	MW(WORD_WEAK := MesBlock_Temp[2][1], 	WORD_STRONG:= MesBlock_Temp[2][2], VAR_OUT:= MesDataExd.MesData.MesU12);		
	MW(WORD_WEAK := MesBlock_Temp[2][3], 	WORD_STRONG:= MesBlock_Temp[2][4], VAR_OUT:= MesDataExd.MesData.MesU23);
	MW(WORD_WEAK := MesBlock_Temp[2][5], 	WORD_STRONG:= MesBlock_Temp[2][6], VAR_OUT:= MesDataExd.MesData.MesU31);
	MW(WORD_WEAK := MesBlock_Temp[2][7], 	WORD_STRONG:= MesBlock_Temp[2][8], VAR_OUT:= MesDataExd.MesData.MesU);		// Seule donnée valide en monophasée. Il faut d'ailleur inverser les words strongs et word weak quand on passe le settings de triphasé à monophasé . 
	MW(WORD_WEAK := MesBlock_Temp[2][9], 	WORD_STRONG:= MesBlock_Temp[2][10], VAR_OUT:= MesDataExd.MesData.MesV1);
	MW(WORD_WEAK := MesBlock_Temp[2][11], WORD_STRONG := MesBlock_Temp[2][12], VAR_OUT:= MesDataExd.MesData.MesV2);
	MW(WORD_WEAK := MesBlock_Temp[2][13], WORD_STRONG := MesBlock_Temp[2][14], VAR_OUT:= MesDataExd.MesData.MesV3);
	MW(WORD_WEAK := MesBlock_Temp[2][17], WORD_STRONG := MesBlock_Temp[2][18], VAR_OUT:= MesDataExd.MesData.MesV);
	
	MW( WORD_STRONG:= MesBlock_Temp[3][1], 	WORD_WEAK := MesBlock_Temp[3][2], VAR_OUT:= MesDataExd.MesData.MesP1);
	MW( WORD_STRONG:= MesBlock_Temp[3][3], 	WORD_WEAK := MesBlock_Temp[3][4], VAR_OUT:= MesDataExd.MesData.MesP2);
	MW( WORD_STRONG:= MesBlock_Temp[3][5], 	WORD_WEAK := MesBlock_Temp[3][6], VAR_OUT:= MesDataExd.MesData.MesP3);
	MW( WORD_STRONG:= MesBlock_Temp[3][7], 	WORD_WEAK := MesBlock_Temp[3][8], VAR_OUT:= MesDataExd.MesData.MesP);
	
	MW( WORD_STRONG:= MesBlock_Temp[3][9], 	WORD_WEAK := MesBlock_Temp[3][10], VAR_OUT:= MesDataExd.MesData.MesQ1);
	MW( WORD_STRONG:= MesBlock_Temp[3][11], 	WORD_WEAK := MesBlock_Temp[3][12], VAR_OUT:= MesDataExd.MesData.MesQ2);
	MW( WORD_STRONG:= MesBlock_Temp[3][13], 	WORD_WEAK := MesBlock_Temp[3][14], VAR_OUT:= MesDataExd.MesData.MesQ3);
	MW( WORD_STRONG:= MesBlock_Temp[3][15], 	WORD_WEAK := MesBlock_Temp[3][16], VAR_OUT:= MesDataExd.MesData.MesQ);
	MW( WORD_STRONG:= MesBlock_Temp[3][23], 	WORD_WEAK := MesBlock_Temp[3][24], VAR_OUT:= MesDataExd.MesData.MesS);
	
	MW( WORD_STRONG:= MesBlock_Temp[4][1], 	WORD_WEAK := MesBlock_Temp[4][2], VAR_OUT:= MesDataExd.MesData.MesTanPhi);
	MW( WORD_STRONG:= MesBlock_Temp[4][3], 	WORD_WEAK := MesBlock_Temp[4][4], VAR_OUT:= MesDataExd.MesData.MesFreq);
	
	MW2( WORD_STRONG:= MesBlock_Temp[5][3], 	WORD_WEAK := MesBlock_Temp[5][4], VAR_OUT := MesDataExd.MesData.MesEActCons,SIZE:=2,FIX:=3);
	MW2( WORD_STRONG:= MesBlock_Temp[5][7], 	WORD_WEAK := MesBlock_Temp[5][8], VAR_OUT := MesDataExd.MesData.MesEActProd,SIZE:=2,FIX:=3);
	MW2( WORD_STRONG:= MesBlock_Temp[5][19], 	WORD_WEAK := MesBlock_Temp[5][20], VAR_OUT := MesDataExd.MesData.MesEReactProd,SIZE:=2,FIX:=3);
	MW2( WORD_STRONG:= MesBlock_Temp[5][23], 	WORD_WEAK := MesBlock_Temp[5][24], VAR_OUT := MesDataExd.MesData.MesEReactCons,SIZE:=2,FIX:=3);
	
	
	//MW( WORD_STRONG:= MesBlock_Temp[4][3], 	WORD_WEAK := MesBlock_Temp[4][4],	SIGNED:=TRUE, FIX:=0 , SIZE:=2, VAR_OUT := MesDataExd.MesData.MesFreq);
	//MW( WORD_STRONG:= MesBlock_Temp[5][1], 	WORD_WEAK := MesBlock_Temp[5][2],	SIGNED:=TRUE, FIX:=0 , SIZE:=2, VAR_OUT := MesDataExd.MesData.MesEActProd);
	//MW( WORD_STRONG:= MesBlock_Temp[5][3], 	WORD_WEAK := MesBlock_Temp[5][4],	SIGNED:=TRUE, FIX:=0 , SIZE:=2, VAR_OUT := MesDataExd.MesData.MesEActCons);
	//MW( WORD_STRONG:= MesBlock_Temp[5][5], 	WORD_WEAK := MesBlock_Temp[5][6],	SIGNED:=TRUE, FIX:=0 , SIZE:=2, VAR_OUT := MesDataExd.MesData.MesEReactProd);
	//MW( WORD_STRONG:= MesBlock_Temp[5][7], 	WORD_WEAK := MesBlock_Temp[5][8],	SIGNED:=TRUE, FIX:=0 , SIZE:=2, VAR_OUT := MesDataExd.MesData.MesEReactCons);
END_IF
END_METHOD

END_FUNCTION_BLOCK

// ---- 01_Equipement_Library/Datalogger/FB_Datalogger_PPCVerrerie.TcPOU
FUNCTION_BLOCK FB_Datalogger_PPCVerrerie	EXTENDS FB_Datalogger_Base	// Data from PPC ( MV + HV )
VAR_INPUT PERSISTENT
	// Parameters of the Object (instance specific) 
	ParamTempoComAlarm			: TIME 			:= T#10S ; 						// (s) Config : Tempo to detect LOC Alarm
	{attribute 'OPC.UA.DA' := '1'} 
	ParamClockReadTime 			: TIME 			:= TIME#200MS;	  				// (Time) Read Modbus Frequency.  
	ParamTimeout				: TIME  		:= T#2S ;			  			// (Time) Timeout for modbus reading
	ParamIPAdr : STRING := '192.168.1.2'; // IP Address for Modbus Requests 
END_VAR
VAR_INPUT
	IN_CmdToggleRead			: BOOL ;
	IN_CmdReset_L				: BOOL  ; // Reset Order .
	
	MesDataExd	AT %Q*				: Datalogger_PPCVerrerie;
	
END_VAR
VAR

	
	//M_ALARMMANAGEMENT VARIABLES//
	TON_ComAlarm				: TON ; 												// Tempo before detecting loss of communication. 
	TON_ComWarning				: TON ; 												// Tempo before detecting loss of one frame.   
	
	MesComWarning				: BOOL ; 												// True if bad communication .
	
	// M_EXECUTE VARIABLES //
	
	TP1							: TP ; 												// (NA) Tempo to define Modbus Reading Frequency  
	
    Trig_Cmd_Read				: R_TRIG;                       

	// Modbus Read Variables
	
	FB_ModbusReadAI : ARRAY[1..2] OF FB_ModbusRead;
	FB_ModbusReadDI : ARRAY[1..2] OF FB_ModbusReadCoils;
	
	ClockRead					AT %Q*		: BOOL ;
	
	// Temp Blocks Filled by Requests
	
	AI_List_1 				: ARRAY[1..128] OF WORD;
	AI_List_2 				: ARRAY[1..128] OF WORD;
	DI_List_1 				: ARRAY[1..2048] OF BOOL;
	DI_List_2 				: ARRAY[1..2048] OF BOOL;
	
	
	
END_VAR

METHOD M_AlarmManagement : BOOL
VAR_INPUT
END_VAR
//////////////////
// Digiware measurement tool alarm and warning management
/////////////////

VAR 
	// Method local variables (reinitialized at each cycle) 
	FB_AlarmCodeManager			: FB_AlarmCodeManager ; 
	
	ComWarning					: BOOL;			// Error in one of the Modbus Requests
	ComAlarm					: BOOL;			// Error in all Modbus Requests
	
END_VAR
ComWarning 	:= FB_ModbusReadAI[1].ModbusReadAlarm OR FB_ModbusReadAI[2].ModbusReadAlarm OR FB_ModbusReadDI[1].ModbusReadAlarm OR FB_ModbusReadDI[2].ModbusReadAlarm;
ComAlarm 	:= FB_ModbusReadAI[1].ModbusReadAlarm AND FB_ModbusReadAI[2].ModbusReadAlarm AND FB_ModbusReadDI[1].ModbusReadAlarm AND FB_ModbusReadDI[2].ModbusReadAlarm;
	
TON_ComAlarm(IN:= ComAlarm , PT:= ParamTempoComAlarm, Q= MesDataExd.MesData.MesAlarmCom) ;	
TON_ComWarning(IN:= ComWarning  , PT:= ParamTempoComAlarm, Q=>MesComWarning) ;

//	General com alarm : All the read FB fucked up


// ALARM CODES //
	FB_AlarmCodeManager(
		bAlarm1			:= MesDataExd.MesData.MesAlarmCom , 						// Communication Alarm #COM
		bAlarm2			:= MesDataExd.MesData.Transfo_225kV.MesWarning_TempLevel1,	// Transfo_225kV : Img Therm 1
		bAlarm3			:= MesDataExd.MesData.Transfo_225kV.MesWarning_TempLevel2,	// Transfo_225kV : Img Therm 2
		bAlarm4			:= MesDataExd.MesData.Transfo_225kV.MesDataExd.MesData.MesAlarmTemp,	// Transfo_225kV : Trigger Temp Oil
		bAlarm5			:= MesDataExd.MesData.Transfo_225kV.MesAlarm_TapChanger ,	// Transfo 225kV : Defaillance Regleur
		bAlarm6			:= MesDataExd.MesData.Mes20kVCourNeutCuveTempTrigger,		// 20 kV Courant Neutre Cuve : Temp Trigger
		bAlarm7			:= MesDataExd.MesData.Mes20kVCourNeutCuveGazDischarge,		// 20 kV Courant Neutre Cuve : Gaz Discharge
		bAlarm8			:= MesDataExd.MesData.Mes20kVCourNeutCuvePressure,			// 20 kV Courant Neutre Cuve : Pressure
		bAlarm9			:= MesDataExd.MesData.Transfo_225kV.MesDataExd.MesData.MesAlarmGas,	// Transfo 225kV : Trigger BuchHolz
		bAlarm10		:= MesDataExd.MesData.Transfo_225kV.MesTrigger_Deletion,	// Transfo_225kV : Trigger Deletion
		bAlarm11		:= MesDataExd.MesData.Transfo_225kV.MesAlarm_OilLevel,      // Transfo_225kV : Alarm Oil level
		bAlarm12		:= MesDataExd.MesData.DS.MesAlarmState,          		// DS : Doors Open          
		bAlarm13		:= MesDataExd.MesData.FSS.MesAlarmFire,			        // FSS : Fire Alarm
		bAlarm14		:= MesDataExd.MesData.MesLocalRemoteOperation, 			// Local/Remote Operation
		bAlarm15		:= MesDataExd.MesData.ES.MesAlarmState,         	 	// ES : Emergency Stop			 
		wAlarmCode		=>MesDataExd.MesData.MesAlarmCode1);

	FB_AlarmCodeManager(	
		bAlarm1			:= MesDataExd.MesData.ProtectRelay_Transfo225kV.MesAlarm_DiscordSectLigneHTB,	//	ProtectRelay_Transfo_225kV :	Alarm Discord Sect Ligne HTB
		bAlarm2			:= MesDataExd.MesData.ProtectRelay_Transfo225kV.MesAlarm_DiscordSectMaltHTB ,   //  ProtectRelay_Transfo_225kV : Alarm Discord Sect Malt HTB 
		bAlarm3			:= MesDataExd.MesData.ProtectRelay_Transfo225kV.MesAlarm_DiscordSectDisjHTB ,   //  ProtectRelay_Transfo_225kV : Alarm Discord Sect Disj HTB 
		bAlarm4			:= MesDataExd.MesData.ProtectRelay_Transfo225kV.MesAlarm_TeleCondamne       ,   //  ProtectRelay_Transfo_225kV : Alarm Tele Condamne       
		bAlarm5			:= MesDataExd.MesData.ProtectRelay_Transfo225kV.MesAlarm_DeTeleCondamne     ,   //  ProtectRelay_Transfo_225kV : Alarm DeTele Condamne     
		bAlarm6			:= MesDataExd.MesData.ProtectRelay_Transfo225kV.MesAlarm_DiscordTeleCondamne,   //  ProtectRelay_Transfo_225kV : Alarm Discord Tele Condamne
		bAlarm7			:= MesDataExd.MesData.ProtectRelay_Transfo225kV.MesDataExd.MesData.MesAlarmImax        ,   //  ProtectRelay_Transfo_225kV : Alarm Imax
		bAlarm8			:= MesDataExd.MesData.ProtectRelay_Transfo225kV.MesAlarm_IoMaxCoteProd      ,   //  ProtectRelay_Transfo_225kV : Alarm Io Max Cote Prod
		bAlarm9			:= MesDataExd.MesData.ProtectRelay_Transfo225kV.MesDataExd.MesData.MesAlarmUmin        ,   //  ProtectRelay_Transfo_225kV : Alarm U min
		bAlarm10		:= MesDataExd.MesData.ProtectRelay_Transfo225kV.MesDataExd.MesData.MesAlarmUmin_Long   ,   //  ProtectRelay_Transfo_225kV : Alarm U min Long
		bAlarm11		:= MesDataExd.MesData.ProtectRelay_Transfo225kV.MesAlarmUMax                ,   //  ProtectRelay_Transfo_225kV : Alarm U max
		bAlarm12		:= MesDataExd.MesData.ProtectRelay_Transfo225kV.MesAlarmUMax_Long           ,   //  ProtectRelay_Transfo_225kV : Alarm U max Long
		bAlarm13		:= MesDataExd.MesData.ProtectRelay_Transfo225kV.MesAlarm_PhaseRpt           ,   //  ProtectRelay_Transfo_225kV : Alarm Phase Rpt
		bAlarm14		:= MesDataExd.MesData.ProtectRelay_Transfo225kV.MesAlarm_ImgTherm     		,	//	ProtectRelay_Transfo_225kV : Alarm Img Therm
		bAlarm15		:= MesDataExd.MesData.ProtectRelay_Transfo225kV.MesAlarm_DifferTransfo		,	//  ProtectRelay_Transfo_225kV : Alarm Differ Transfo
		wAlarmCode		=>MesDataExd.MesData.MesAlarmCode2);	


	FB_AlarmCodeManager(	
		bAlarm1			:= MesDataExd.MesData.ProtectRelay_Transfo225kV.MesAlarm_FreqMax ,	// ProtectRelay_Transfo_225kV : Alarm Freq Max
		bAlarm2			:= MesDataExd.MesData.ProtectRelay_Transfo225kV.MesAlarm_FreqMin ,  // ProtectRelay_Transfo_225kV : Alarm Freq Min
		bAlarm3			:= MesDataExd.MesData.MainHVCB.MesDataExd.MesData.MesClosed ,					// MainHVCB : Closed 
		bAlarm4			:= MesDataExd.MesData.MainHVCB.MesAlarm_SF6      ,					// MainHVCB : Alarm SF6
		bAlarm5			:= MesDataExd.MesData.MainHVCB.MesAlarm_Disarmed ,					// MainHVCB : Alarm Disarmed
		bAlarm6			:= MesDataExd.MesData.MainHVCB.MesComutLocal     ,					// MainHVCB : Comut Local
		bAlarm7			:= MesDataExd.MesData.Transfo_225kV.MesTransfoRefrigLocal,    		// Transfo_225kV : Transfo Refrig Local
		bAlarm8			:= MesDataExd.MesData.Transfo_225kV.MesTrigger_NonReturnValve,      // Transfo_225kV : Trigger Non Return Valve
		bAlarm9			:= MesDataExd.MesData.Transfo_225kV.MesTrigger_ProtectRelay,        // Transfo_225kV : Trigger Protect Relay
		bAlarm10		:= MesDataExd.MesData.Transfo_Aux.MesDataExd.MesData.MesAlarmTemp,				// Transfo_Aux : Alarm Temp
		bAlarm11		:= MesDataExd.MesData.Transfo_Aux.MesDataExd.MesData.MesAlarmGas,              // Transfo_Aux : Alarm Gas
		bAlarm12		:= MesDataExd.MesData.Transfo_Aux.MesDataExd.MesData.MesAlarmOilLevel,         // Transfo_Aux : Alarm Pressure
		bAlarm13		:= MesDataExd.MesData.MesAuxTransfoMeltingFusesContact,			// Transfo_Aux : Melting Fuses Contact     
		bAlarm14		:= MesDataExd.MesData.MesAuxTransfoSwitchGear,                     // Transfo_Aux : Transfo Switch Gear
		bAlarm15		:=FALSE,
		wAlarmCode		=>MesDataExd.MesData.MesAlarmCode3);			
		
		
// WARNING CODES //
	FB_AlarmCodeManager(		
		bAlarm1			:=MesComWarning	,				 							// Communication Warning
		bAlarm2			:= MesDataExd.MesData.ProtectRelay_MainHVCB.MesAlarm_Phase1 , 			// ProtectRelay_MainHVCB : Default Phase 1       
		bAlarm3			:= MesDataExd.MesData.ProtectRelay_MainHVCB.MesAlarm_Phase2 , 			// ProtectRelay_MainHVCB : Default Phase 2       
		bAlarm4			:= MesDataExd.MesData.ProtectRelay_MainHVCB.MesAlarm_Phase3 , 			// ProtectRelay_MainHVCB : Default Phase 3       
		bAlarm5			:= MesDataExd.MesData.ProtectRelay_MainHVCB.MesAlarm_PhaseRpt , 		// ProtectRelay_MainHVCB : Default Phase Rpt      
		bAlarm6			:= MesDataExd.MesData.ProtectRelay_MainHVCB.MesAlarm_Ground , 			// ProtectRelay_MainHVCB : Default Phase Ground        
		bAlarm7			:= MesDataExd.MesData.ProtectRelay_MainHVCB.MesAlarm_GroundRpt , 		// ProtectRelay_MainHVCB : Default Phase Ground Rpt     
		bAlarm8			:= MesDataExd.MesData.ProtectRelay_MainHVCB.MesAlarm_MaxUInverse , 		// ProtectRelay_MainHVCB : Default Max U Inverse   
		bAlarm9			:= MesDataExd.MesData.ProtectRelay_MainHVCB.MesAlarm_MaxP , 			// ProtectRelay_MainHVCB : Default Max P
		bAlarm10		:= MesDataExd.MesData.ProtectRelay_MainHVCB.MesAlarm_CB , 				// ProtectRelay_MainHVCB : Default Circuit Breaker
		bAlarm11		:= MesDataExd.MesData.ProtectRelay_MainHVCB.MesAlarm_Watchdog , 		// ProtectRelay_MainHVCB : Default Watchdog     
		bAlarm12		:= MesDataExd.MesData.ProtectRelay_MainHVCB.MesDataExd.MesData.MesAlarmTCS  , 		// ProtectRelay_MainHVCB : Default Major        
		bAlarm13		:= MesDataExd.MesData.ProtectRelay_Transfo225kV.MesAlarm_PhaseRpt ,		// ProtectRelay_Transfo225kV : Default Phase Rpt
		bAlarm14		:= MesDataExd.MesData.ProtectRelay_Transfo225kV.MesAlarm_ImgTherm , 	// ProtectRelay_Transfo225kV : Default img Therm
		bAlarm15		:= MesDataExd.MesData.MainHVCB.MesAlarm_ArmingMotor , 					// MainHVCB : Default Arming Motor
		wAlarmCode		=>MesDataExd.MesData.MesWarningCode1);

	FB_AlarmCodeManager(		
		bAlarm1			:= MesDataExd.MesData.MainHVCB.MesAlarm_230V, 							// MainHVCB : Default Aux 230 Vac				 
		bAlarm2			:= MesDataExd.MesData.MainHVCB.MesAlarmPwr, 							// MainHVCB : Default Alim Bobine
		bAlarm3			:= MesDataExd.MesData.Transfo_225kV.MesWarningGas, 						// Transfo_225kV : Buchholz Gas Warning
		bAlarm4			:= MesDataExd.MesData.Transfo_225kV.MesDataExd.MesData.MesWarningTemp, 			// Transfo_225kV : Temperature Warning
		bAlarm5			:= MesDataExd.MesData.ProtectRelay_Transfo225kV.MesDataExd.MesData.MesAlarmTCS , 	// ProtectRelay_Transfo225kV : Major Default
		bAlarm6			:= MesDataExd.MesData.ProtectRelay_Transfo225kV.MesWarning_ImgTherm , 	// ProtectRelay_Transfo225kV : Warning Img Therm
		bAlarm7			:= MesDataExd.MesData.TapChanger.MesAlarm,								// 225 kV Regleur : Default
		bAlarm8			:= MesDataExd.MesData.TapChanger.MesAlarm_Discordance, 					// 225 kV Regleur : Default Discordance
		bAlarm9			:= MesDataExd.MesData.ProtectRelay_MainMVCB.MesAlarm_Phase1, 			// Protection Relay Main MVCB : Default Phase 1
		bAlarm10		:= MesDataExd.MesData.ProtectRelay_MainMVCB.MesAlarm_Phase2, 			// Protection Relay Main MVCB : Default Phase 2
		bAlarm11		:= MesDataExd.MesData.ProtectRelay_MainMVCB.MesAlarm_CB, 				// Protection Relay Main MVCB : Default Circuit Breaker
		bAlarm12		:=FALSE , 													//
		bAlarm13		:= MesDataExd.MesData.MainMVCB.MesTripped 	, 							// Main MVCB : Tripped
		bAlarm14		:= MesDataExd.MesData.ProtectRelay_MainMVCB.MesDataExd.MesData.MesAlarmTCS , 		// Protection Relay Main MVCB : Alarm TCS
		bAlarm15		:= MesDataExd.MesData.ProtectRelay_MainMVCB.MesDataExd.MesData.MesWatchdog,		// Protection Relay Main MVCB : Watchdog
		wAlarmCode		=>MesDataExd.MesData.MesWarningCode2);		

	FB_AlarmCodeManager(		
		bAlarm1			:= MesDataExd.MesData.ProtectRelay_FeederMVCB[1].MesDataExd.MesData.MesAlarmImax, 							//  ProtectRelay_FeederMVCB Midi Max I Alarm
		bAlarm2			:= MesDataExd.MesData.ProtectRelay_FeederMVCB[1].MesAlarm_MaxP ,								//  ProtectRelay_FeederMVCB Midi Max P Alarm 
		bAlarm3			:= MesDataExd.MesData.ProtectRelay_FeederMVCB[1].MesAlarm_Ground , 								//  ProtectRelay_FeederMVCB Midi Ground Alarm
		bAlarm4			:= MesDataExd.MesData.ProtectRelay_FeederMVCB[1].MesAlarm_CablesOvercharge, 					//	ProtectRelay_FeederMVCB Midi Cables Overcharge
		bAlarm5			:= MesDataExd.MesData.ProtectRelay_FeederMVCB[1].MesAlarm_FaultFrom225kV, 						//  ProtectRelay_FeederMVCB Midi Fault From 225 kV   
		bAlarm6			:= MesDataExd.MesData.ProtectRelay_FeederMVCB[1].MesDataExd.MesData.MesAlarmTCS , 							//  ProtectRelay_FeederMVCB Midi Default Major       
		bAlarm7			:= MesDataExd.MesData.ProtectRelay_FeederMVCB[2].MesDataExd.MesData.MesAlarmImax, 	 						//  ProtectRelay_FeederMVCB Plat Max I Alarm      
		bAlarm8			:= MesDataExd.MesData.ProtectRelay_FeederMVCB[2].MesAlarm_MaxP ,			     				//  ProtectRelay_FeederMVCB Plat Max P Alarm        
		bAlarm9			:= MesDataExd.MesData.ProtectRelay_FeederMVCB[2].MesAlarm_Ground , 		   						//  ProtectRelay_FeederMVCB Plat Ground Alarm          
		bAlarm10		:= MesDataExd.MesData.ProtectRelay_FeederMVCB[2].MesAlarm_CablesOvercharge, 					//  ProtectRelay_FeederMVCB Plat Cables Overcharge 
		bAlarm11		:= MesDataExd.MesData.ProtectRelay_FeederMVCB[2].MesAlarm_FaultFrom225kV, 	 					//  ProtectRelay_FeederMVCB Plat Fault From 225 kV    
		bAlarm12		:= MesDataExd.MesData.ProtectRelay_FeederMVCB[2].MesDataExd.MesData.MesAlarmTCS,				 			//  ProtectRelay_FeederMVCB Plat Default Major                  
		bAlarm13		:=FALSE,   //
		bAlarm14		:=FALSE,   //
		bAlarm15		:=FALSE,   //
		wAlarmCode		=>MesDataExd.MesData.MesWarningCode3);

	FB_AlarmCodeManager(		
		bAlarm1			:= MesDataExd.MesData.Mes20kVCourNeutCuveDefaultMasseCuve1,			//	 20 kV Courant Neutre Cuve Default Masse 1
		bAlarm2			:= MesDataExd.MesData.Mes20kVCourNeutCuveDefaultMasseCuve2,			//	 20 kV Courant Neutre Cuve Default Masse 2
		bAlarm3			:= MesDataExd.MesData.Mes20kVCourNeutCuveDefaultGround,				//	 20 kV Courant Neutre Cuve Default Ground 
		bAlarm4			:= MesDataExd.MesData.Mes20kVCourNeutCuveTempAlarm,					//	 20 kV Courant Neutre Cuve Temp  
		bAlarm5			:= MesDataExd.MesData.MesAuxBt400VDefaultPermut, 					//	 Aux Bt 400 V  : Default Permut 
		bAlarm6			:= MesDataExd.MesData.UPS_CE.MesAlarm_Batt, 			      		//	 UPC CE : Default Batt
		bAlarm7			:= MesDataExd.MesData.UPS_CE.MesDataExd.MesData.MesAlarmState, 				//	 UPC CE : Default Redress
		bAlarm8			:= MesDataExd.MesData.UPS_CE.MesAlarm_IsolBatt,		    			//   UPC CE : Default Isol Batt
		bAlarm9			:= MesDataExd.MesData.UPS_TCM.MesAlarm_Batt,			      		//   UPC TCM : Default Batt
		bAlarm10		:= MesDataExd.MesData.UPS_TCM.MesDataExd.MesData.MesAlarmState,	 			//	 UPC TCM : Default Redress
		bAlarm11		:= MesDataExd.MesData.MesAuxBtDefaultInverter, 						//	 Aux Bt : Default Inverter
		bAlarm12		:= MesDataExd.MesData.MesAuxBtSyntDefaultDistrib48VccJdb, 			//	 Aux Bt Synt : Default Distrib 48 Vcc Jdb
		bAlarm13		:= MesDataExd.MesData.MesAuxBtSyntDefaultDistrib48VccLocker, 		//	 Aux Bt Synt : Default Distrib 48 Vcc Locker
		bAlarm14		:=FALSE, //
		bAlarm15		:=FALSE, //
		wAlarmCode		=>MesDataExd.MesData.MesWarningCode4);		
		
	FB_AlarmCodeManager(		
		bAlarm1			:= MesDataExd.MesData.Mes20kVCourNeutCuveMaxIexp2,	//	 20 kV Courant Neutre Cuve Default Max I Exp 2
		bAlarm2			:= MesDataExd.MesData.Mes20kVCourNeutCuveMaxIexp4,  //	 20 kV Courant Neutre Cuve Default Max I Exp 4
		bAlarm3			:= MesDataExd.MesData.Mes20kVCourNeutCuveMaxI0exp4, //	 20 kV Courant Neutre Cuve Default Max I0 Exp 4
		bAlarm4			:= MesDataExd.MesData.ProtectRelay_FeederMVCB[1].MesDataExd.MesData.MesTripped, // ProtectRelay_FeederMVCB Midi Tripped
		bAlarm5			:= MesDataExd.MesData.ProtectRelay_FeederMVCB[2].MesDataExd.MesData.MesTripped, // ProtectRelay_FeederMVCB Plat Tripped
		bAlarm6			:= MesDataExd.MesData.MesAuxHTSect225kV		,					//	Aux HT : Sect 225 kV
		bAlarm7			:= MesDataExd.MesData.MesAuxHtSmaltHTBOpen	,                   //	Aux HT : Malt HTB Open
		bAlarm8			:= MesDataExd.MesData.MesAuxHtFusionFuseMeasures225kV	,       //	Aux HT : Fusion Fuse Measures 225 kV
		bAlarm9			:= MesDataExd.MesData.MesAuxHtFusionFuseProtect225kV	,       //  Aux HT : Fusion Fuse Protect 225 kV
		bAlarm10		:= MesDataExd.MesData.MesAuxHtFusionFuseCountRte225kV	,       //	Aux HT : Fusion Fuse Count Rte 225 kV
		bAlarm11		:= MesDataExd.MesData.MesAuxHtShortCircuitCurrentProtectCcp2,   //  Aux HT : Short Circuit Current Protect Ccp2
		bAlarm12		:= MesDataExd.MesData.MesAuxHtDisjCount20kVOpen		,           //	Aux HT : Disj Count 20kV Open
		bAlarm13		:= MesDataExd.MesData.MesAuxHtDisjRefVoltage20kVOpen,			//  Aux HT : Disj Ref Voltage 20kV Open
		bAlarm14		:= MesDataExd.MesData.MesAuxHtShortCircuitCurrentProtectCcp3, 	//	Aux HT : Short Circuit Current Protect Ccp3
		bAlarm15		:= MesDataExd.MesData.MesAuxBtTriggerGeneralDisj, 				//  Aux BT : Trigger General Disj
		wAlarmCode		=>MesDataExd.MesData.MesWarningCode5);
		
	FB_AlarmCodeManager(		
		bAlarm1			:= MesDataExd.MesData.Mes20kVCourNeutCuveMaxIexp2,	//	 20 kV Courant Neutre Cuve Default Max I Exp 2
		bAlarm2			:= MesDataExd.MesData.Mes20kVCourNeutCuveMaxIexp4,  //	 20 kV Courant Neutre Cuve Default Max I Exp 4
		bAlarm3			:= MesDataExd.MesData.Mes20kVCourNeutCuveMaxI0exp4, //	 20 kV Courant Neutre Cuve Default Max I0 Exp 4
		bAlarm4			:= MesDataExd.MesData.ProtectRelay_FeederMVCB[1].MesDataExd.MesData.MesTripped, // ProtectRelay_FeederMVCB Midi Tripped
		bAlarm5			:= MesDataExd.MesData.ProtectRelay_FeederMVCB[2].MesDataExd.MesData.MesTripped, // ProtectRelay_FeederMVCB Plat Tripped
		bAlarm6			:= MesDataExd.MesData.MesAuxHTSect225kV		,					//	Aux HT : Sect 225 kV
		bAlarm7			:= MesDataExd.MesData.MesAuxHtSmaltHTBOpen	,                   //	Aux HT : Malt HTB Open
		bAlarm8			:= MesDataExd.MesData.MesAuxHtFusionFuseMeasures225kV	,       //	Aux HT : Fusion Fuse Measures 225 kV
		bAlarm9			:= MesDataExd.MesData.MesAuxHtFusionFuseProtect225kV	,       //  Aux HT : Fusion Fuse Protect 225 kV
		bAlarm10		:= MesDataExd.MesData.MesAuxHtFusionFuseCountRte225kV	,       //	Aux HT : Fusion Fuse Count Rte 225 kV
		bAlarm11		:= MesDataExd.MesData.MesAuxHtShortCircuitCurrentProtectCcp2,   //  Aux HT : Short Circuit Current Protect Ccp2
		bAlarm12		:= MesDataExd.MesData.MesAuxHtDisjCount20kVOpen		,           //	Aux HT : Disj Count 20kV Open
		bAlarm13		:= MesDataExd.MesData.MesAuxHtDisjRefVoltage20kVOpen,			//  Aux HT : Disj Ref Voltage 20kV Open
		bAlarm14		:= MesDataExd.MesData.MesAuxHtShortCircuitCurrentProtectCcp3, 	//	Aux HT : Short Circuit Current Protect Ccp3
		bAlarm15		:= MesDataExd.MesData.MesAuxBtTriggerGeneralDisj, 				//  Aux BT : Trigger General Disj
		wAlarmCode		=>MesDataExd.MesData.MesWarningCode6);
		
		
// EVENT CODE //
	FB_AlarmCodeManager(
		bAlarm1			:= MesDataExd.MesData.MesAuxBt400VManqueAC			 ,  		// Aux BT 400 V : Manque AC     
		bAlarm2			:= MesDataExd.MesData.MesAuxBt400VDecltAntenneScada	 ,  		// Aux BT 400 V : Declt Antenne Scada
		bAlarm3			:= MesDataExd.MesData.MesAuxBt400VDecltAntennePrio	 ,  		// Aux BT 400 V : Declt Antenne Prio
		bAlarm4			:= MesDataExd.MesData.MesAuxBt400VVoltageLossNormalAlim	, 		// Aux BT 400 V : Voltage Loss Normal Alim
		bAlarm5			:= MesDataExd.MesData.MesAuxBt400VVoltageLossSecoursAlim,   	// Aux BT 400 V : Voltage Loss Secours Alim
		bAlarm6			:= MesDataExd.MesData.MesAuxBt400VDefaultPermut	,           	// Aux BT 400 V : Default Permut 
		bAlarm7			:= MesDataExd.MesData.TapChanger.MesModeAuto, 					// 225 kV Regleur :	Mode Auto
		bAlarm8			:= MesDataExd.MesData.TapChanger.MesModeManual,                 // 225 kV Regleur :	Mode Manual                                                                                                                                                                                              
		bAlarm9			:= MesDataExd.MesData.TapChanger.MesState_ManoeuverAuthorized, 	// 225 kV Regleur :	State Manoeuver Authorized
		bAlarm10		:= MesDataExd.MesData.TapChanger.MesAlarm_NoOutletDetected, 	// 225 kV Regleur :	No Outlet Detected	
		bAlarm11		:= MesDataExd.MesData.ProtectRelay_MainHVCB.OUT_CmdOpen , 		// ProtectRelay_MainHVCB : Cmd Open
		bAlarm12		:= MesDataExd.MesData.ProtectRelay_MainHVCB.OUT_CmdClose,       // ProtectRelay_MainHVCB : Cmd Close
		bAlarm13		:= MesDataExd.MesData.ProtectRelay_MainMVCB.OUT_CmdOpen ,       // ProtectRelay_MainMVCB : Cmd Open
		bAlarm14		:= MesDataExd.MesData.ProtectRelay_MainMVCB.OUT_CmdClose,       // ProtectRelay_MainMVCB : Cmd Close
		bAlarm15		:=FALSE, 
		wAlarmCode		=>MesDataExd.MesData.MesEventCode1);
	
	FB_AlarmCodeManager(	
		bAlarm1			:= MesDataExd.MesData.ProtectRelay_FeederMVCB[1].OUT_CmdOpen , 	// ProtectRelay_FeederMVCB Midi : Cmd Open
		bAlarm2			:= MesDataExd.MesData.ProtectRelay_FeederMVCB[1].OUT_CmdClose,     // ProtectRelay_FeederMVCB Midi  : Cmd Close
		bAlarm3			:= MesDataExd.MesData.ProtectRelay_FeederMVCB[2].OUT_CmdOpen  ,    // ProtectRelay_FeederMVCB Plat  : Cmd Open
		bAlarm4			:= MesDataExd.MesData.ProtectRelay_FeederMVCB[2].OUT_CmdClose ,	// ProtectRelay_FeederMVCB Plat  : Cmd Close
		bAlarm5			:= MesDataExd.MesData.TapChanger.OUT_CmdRampUp,					// 225 kV Regleur : Cmd Ramp Up
		bAlarm6			:= MesDataExd.MesData.TapChanger.OUT_CmdRampDown ,                 // 225 kV Regleur :	Cmd Ramp Down
		bAlarm7			:= MesDataExd.MesData.MesAuxHtOpenSectLine225kV	 ,				// Aux Ht : Sect Line 225 kV Open
		bAlarm8			:= MesDataExd.MesData.MesAuxHtCloseSectLine225kV	,               // Aux Ht : Sect Line 225 kV Close
		bAlarm9			:= MesDataExd.MesData.MesAuxHtTeleCondamnSl225kV	 ,				// Aux Ht : Tele Condamn Sl 225 kV 
		bAlarm10		:= MesDataExd.MesData.MesAuxHtDeTeleCondamnSl225kV,       		// Aux Ht : DeTele Condamn Sl 225 kV
		bAlarm11		:= MesDataExd.MesData.MesAuxHtTelecommandeRelestActif ,			// Aux Ht : Telecommande Relest Actif
		bAlarm12		:= MesDataExd.MesData.MesAuxHtTelecommandeRelestPassif,           // Aux Ht : Telecommande Relest Passif
		bAlarm13		:= FALSE,
		bAlarm14		:= FALSE,
		bAlarm15		:= FALSE,
		wAlarmCode		=>MesDataExd.MesData.MesEventCode2);	
		
		
	FB_AlarmCodeManager(
		bAlarm1			:= MesDataExd.MesData.MesAuxHtOpenSectMalt,				// Aux Ht Sect Malt : Open
		bAlarm2			:= MesDataExd.MesData.MesAuxHtCloseSectMalt,				// Aux Ht Sect Malt : Close
		bAlarm3			:= MesDataExd.MesData.MesAuxBtSyntOpenDistrib48VccJdb,		// Aux Bt Synt : Open Distrib 48 Vcc Jdb
		bAlarm4			:= MesDataExd.MesData.MesAuxBtSyntOpenDistrib48VccLocker,	// Aux Bt Synt : Open Distrib 48 Vcc Locker
		bAlarm5			:= MesDataExd.MesData.MesAuxBt400VPermutAutoStopMode	,	// Aux Bt 400 V Permut Auto Stop Mode				
		bAlarm6			:= MesDataExd.MesData.MesAuxBt400VPermutAutoNormalMode	 ,	// Aux Bt 400 V Permut Auto Normal Mode
		bAlarm7			:= MesDataExd.MesData.MesAuxBt400VPermutAutoSecoursMode,	// Aux Bt 400 V Permut Auto Secours Mode
		bAlarm8			:= MesDataExd.MesData.MesAuxBt400VPermutModeAuto	,		// Aux Bt 400 V Permut Mode Auto
		bAlarm9			:= MesDataExd.MesData.UPS_CE.MesOpened_CBRectifier	,		// UPC CE : Opened CB Rectifier
		bAlarm10		:= MesDataExd.MesData.UPS_CE.MesOpened_CBBatt		    ,	// UPC CE : Opened CB Batt
		bAlarm11		:= MesDataExd.MesData.UPS_CE.MesOpened_CBAntenna		 ,	// UPC CE : Opened CB Antenna
		bAlarm12		:= MesDataExd.MesData.UPS_TCM.MesOpened_CBRectifier	,	// UPC TCM : Opened CB Rectifier
		bAlarm13		:= MesDataExd.MesData.UPS_TCM.MesOpened_CBBatt	   	 ,		// UPC TCM : Opened CB Batt
		bAlarm14		:= MesDataExd.MesData.UPS_TCM.MesOpened_CBAntenna	  ,		// UPC TCM : Opened CB Antenna 
		bAlarm15		:= FALSE,//  
		wAlarmCode		=>MesDataExd.MesData.MesEventCode3);
END_METHOD

METHOD M_CP
//////////////////
//  Emulator
/////////////////

VAR 
	// Method local variables (reinitialized at each cycle) 
	

END_VAR


SUPER^.M_CP() ; 




Trig_Cmd_Read(CLK:=IN_CmdToggleRead);
Trig_Cmd_Write(CLK:=IN_CmdToggleWrite);
	
IF Trig_Cmd_Read.Q THEN
	IN_CmdToggleRead := FALSE;
	MesDataExd.MesData.MesCP_Read := NOT MesDataExd.MesData.MesCP_Read;
END_IF


IF Trig_Cmd_Write.Q THEN
	IN_CmdToggleWrite := FALSE;
	MesDataExd.MesData.MesCP_Write := NOT MesDataExd.MesData.MesCP_Write;
END_IF
END_METHOD

METHOD M_Execute
//////////////////
//  Method Calls 
/////////////////
VAR 
	// Method local variables (reinitialized at each cycle) 
	// EMULATOR

	
END_VAR
// READING AND WRITING CLOCK //
	TP1(IN:=NOT TP1.Q , PT:= ParamClockReadTime);
	ClockRead 		:= TP1.Q;
	
// METHODS CALLS //

	M_Read() ; 
	M_CP();
	
// EVALUATE  /////////////
	

	
	////////////////////
	M_AlarmManagement();
END_METHOD

METHOD M_Read : BOOL
VAR_INPUT
END_VAR
VAR
	MW					: FB_MergeWordsToDint;
END_VAR
// CP-Read / Write 


IF MesDataExd.MesData.MesCP_Read  THEN	

	// Analogic Inputs Modbus Requests
	
	FB_ModbusReadAI[1](pDestAddr := ADR(AI_List_1),
					sIPAddr := ParamIPAdr,
					tTimeout := ParamTimeout,
					nTcpPort := 502,
					nQuantity := 123,
					nMBAddr := 593,
					cbLength := SIZEOF(AI_List_1),
					nUnitID := 1,
					ClockRead := ClockRead,
					Reset := IN_CmdReset_L);
					
	FB_ModbusReadAI[2](pDestAddr := ADR(AI_List_2),
					sIPAddr := ParamIPAdr,
					tTimeout := ParamTimeout,
					nTcpPort := 502,
					nQuantity := 97,
					nMBAddr := 721,
					cbLength := SIZEOF(AI_List_2),
					nUnitID := 1,
					ClockRead := ClockRead,
					Reset := IN_CmdReset_L);
					
	// Digital Inputs Modbus Requests 
	
	FB_ModbusReadDI[1](pDestAddr := ADR(DI_List_1),
					sIPAddr := ParamIPAdr,
					tTimeout := ParamTimeout,
					nTcpPort := 502,
					nQuantity := 1683,
					nMBAddr := 480,
					cbLength := SIZEOF(DI_List_1),
					nUnitID := 1,
					ClockRead := ClockRead,
					Reset := IN_CmdReset_L);
					
	FB_ModbusReadDI[2](pDestAddr := ADR(DI_List_2),
					sIPAddr := ParamIPAdr,
					tTimeout := ParamTimeout,
					nTcpPort := 502,
					nQuantity := 1249,
					nMBAddr := 5072,
					cbLength := SIZEOF(DI_List_2),
					nUnitID := 1,
					ClockRead := ClockRead,
					Reset := IN_CmdReset_L);
	
					
					
	//  MesDataExd.MesData.Filling Digital Data				
	
	MesDataExd.MesData.ProtectRelay_MainHVCB.MesAlarm_Phase1			:= DI_List_1[1]   ;
	MesDataExd.MesData.ProtectRelay_MainHVCB.MesAlarm_Phase2		    := DI_List_1[2]   ;
	MesDataExd.MesData.ProtectRelay_MainHVCB.MesAlarm_Phase3			:= DI_List_1[3]   ;
	MesDataExd.MesData.ProtectRelay_MainHVCB.MesAlarm_PhaseRpt			:= DI_List_1[33]  ;
	MesDataExd.MesData.ProtectRelay_MainHVCB.MesAlarm_Ground			:= DI_List_1[35]  ;
	MesDataExd.MesData.ProtectRelay_MainHVCB.MesAlarm_GroundRpt		:= DI_List_1[36]  ;
	MesDataExd.MesData.ProtectRelay_MainHVCB.MesAlarm_MaxUInverse		:= DI_List_1[37]  ;
	MesDataExd.MesData.ProtectRelay_MainHVCB.MesAlarm_MaxP				:= DI_List_1[38]  ;
	MesDataExd.MesData.ProtectRelay_MainHVCB.MesAlarm_CB				:= DI_List_1[39]  ;	
	MesDataExd.MesData.ProtectRelay_MainHVCB.MesAlarm_Watchdog			:= DI_List_1[148] ;
	
				
	MesDataExd.MesData.ProtectRelay_Transfo225kV.MesAlarm_DiscordSectLigneHTB		   := DI_List_1[164]    ;
	MesDataExd.MesData.ProtectRelay_Transfo225kV.MesAlarm_DiscordSectMaltHTB         := DI_List_1[165]    ;
	MesDataExd.MesData.ProtectRelay_Transfo225kV.MesAlarm_DiscordSectDisjHTB         := DI_List_1[166]    ;
	MesDataExd.MesData.ProtectRelay_Transfo225kV.MesAlarm_TeleCondamne               := DI_List_1[167]    ;
	MesDataExd.MesData.ProtectRelay_Transfo225kV.MesAlarm_DeTeleCondamne             := DI_List_1[168]    ;
	MesDataExd.MesData.ProtectRelay_Transfo225kV.MesAlarm_DiscordTeleCondamne	       := DI_List_1[169]    ;
	MesDataExd.MesData.ProtectRelay_Transfo225kV.MesDataExd.MesData.MesAlarmImax                := DI_List_1[171]    ;
	MesDataExd.MesData.ProtectRelay_Transfo225kV.MesAlarm_IoMaxCoteProd              := DI_List_1[172]    ;
	MesDataExd.MesData.ProtectRelay_Transfo225kV.MesDataExd.MesData.MesAlarmUmin                := DI_List_1[173]    ;
	MesDataExd.MesData.ProtectRelay_Transfo225kV.MesDataExd.MesData.MesAlarmUmin_Long           := DI_List_1[174]    ;
	MesDataExd.MesData.ProtectRelay_Transfo225kV.MesAlarmUMax                        := DI_List_1[175]    ;
	MesDataExd.MesData.ProtectRelay_Transfo225kV.MesAlarmUMax_Long                   := DI_List_1[176]    ;
	MesDataExd.MesData.ProtectRelay_Transfo225kV.MesAlarm_PhaseRpt           	 	   := DI_List_1[177]    ;
	MesDataExd.MesData.ProtectRelay_Transfo225kV.MesWarning_ImgTherm                 := DI_List_1[178]    ;
	MesDataExd.MesData.ProtectRelay_Transfo225kV.MesAlarm_ImgTherm                   := DI_List_1[179]    ;
	MesDataExd.MesData.ProtectRelay_Transfo225kV.MesAlarm_DifferTransfo              := DI_List_1[180]    ;
	MesDataExd.MesData.ProtectRelay_Transfo225kV.MesAlarm_FreqMax                    := DI_List_1[181]    ;
	MesDataExd.MesData.ProtectRelay_Transfo225kV.MesAlarm_FreqMin                    := DI_List_1[183]    ;
	
	
	MesDataExd.MesData.MainHVCB.MesDataExd.MesData.MesClosed            				:= DI_List_1[193]    ;
	MesDataExd.MesData.MainHVCB.MesAlarm_SF6              				:= DI_List_1[197]    ;
	MesDataExd.MesData.MainHVCB.MesAlarm_Disarmed             	 		:= DI_List_1[198]    ;
	MesDataExd.MesData.MainHVCB.MesComutLocal         			   		:= DI_List_1[199]    ;
	MesDataExd.MesData.MainHVCB.MesAlarm_ArmingMotor           			:= DI_List_1[200]    ;
	MesDataExd.MesData.MainHVCB.MesAlarm_230V           					:= DI_List_1[201]    ;
	MesDataExd.MesData.MainHVCB.MesAlarmPwr          			 			:= DI_List_1[202]    ;
	
	MesDataExd.MesData.Transfo_225kV.MesWarningGas               			:= DI_List_1[220]    ;
	MesDataExd.MesData.Transfo_225kV.MesDataExd.MesData.MesAlarmGas           	 	:= DI_List_1[221]    ;
	MesDataExd.MesData.Transfo_225kV.MesDataExd.MesData.MesWarningTemp               := DI_List_1[222]    ;
	MesDataExd.MesData.Transfo_225kV.MesDataExd.MesData.MesAlarmGas             		:= DI_List_1[223]    ;
	MesDataExd.MesData.Transfo_225kV.MesWarning_TempLevel1           		:= DI_List_1[224]    ;
	MesDataExd.MesData.Transfo_225kV.MesWarning_TempLevel2          		:= DI_List_1[225]    ;
	MesDataExd.MesData.Transfo_225kV.MesTrigger_Deletion            		:= DI_List_1[228]    ;
	MesDataExd.MesData.Transfo_225kV.MesAlarm_OilLevel              		:= DI_List_1[229]    ;
	MesDataExd.MesData.Transfo_225kV.MesTransfoRefrigLocal                := DI_List_1[230]    ;
	MesDataExd.MesData.Transfo_225kV.MesTrigger_NonReturnValve       		:= DI_List_1[231]    ;
	MesDataExd.MesData.Transfo_225kV.MesTrigger_ProtectRelay      		:= DI_List_1[232]    ;
	MesDataExd.MesData.Transfo_225kV.MesAlarm_TapChanger            		:= DI_List_1[233]    ;
	
	MesDataExd.MesData.Mes20kVCourNeutCuveDefaultMasseCuve1		:= DI_List_1[305]	;
	MesDataExd.MesData.Mes20kVCourNeutCuveMaxIexp2				:= DI_List_1[306]   ;
	MesDataExd.MesData.Mes20kVCourNeutCuveDefaultMasseCuve2  		:= DI_List_1[307]   ;
	MesDataExd.MesData.Mes20kVCourNeutCuveMaxIexp4				:= DI_List_1[308]   ;
	MesDataExd.MesData.Mes20kVCourNeutCuveDefaultGround	    	:= DI_List_1[309]   ;
	MesDataExd.MesData.Mes20kVCourNeutCuveMaxI0exp4		    	:= DI_List_1[310]   ;
	MesDataExd.MesData.Mes20kVCourNeutCuveTempAlarm		    	:= DI_List_1[439]   ;
	MesDataExd.MesData.Mes20kVCourNeutCuveTempTrigger				:= DI_List_1[440]   ;
	MesDataExd.MesData.Mes20kVCourNeutCuveGazDischarge			:= DI_List_1[441]   ;
	MesDataExd.MesData.Mes20kVCourNeutCuvePressure           		:= DI_List_1[442]   ;
	
	MesDataExd.MesData.ProtectRelay_MainMVCB.MesAlarm_Phase1 			:= DI_List_1[457]	;
	MesDataExd.MesData.ProtectRelay_MainMVCB.MesAlarm_Phase2			:= DI_List_1[459]   ; // Phase 3  ? 
	MesDataExd.MesData.ProtectRelay_MainMVCB.MesAlarm_CB 				:= DI_List_1[495]   ;
	MesDataExd.MesData.ProtectRelay_MainMVCB.MesDataExd.MesData.MesTripped 		:= DI_List_1[586]   ; // Mes20kVGeneralHVCellProtectCircuitBreaker
	 /  MesDataExd.MesData.Mes20kVGeneralHVCellDefaultFrom225kV			:= DI_List_1[592]   ;
	
	MesDataExd.MesData.ProtectRelay_FeederMVCB[1].MesDataExd.MesData.MesAlarmImax 							:=	DI_List_1[609]	;
	MesDataExd.MesData.ProtectRelay_FeederMVCB[1].MesAlarm_MaxP									:=	DI_List_1[611]  ;
	MesDataExd.MesData.ProtectRelay_FeederMVCB[1].MesAlarm_Ground									:=	DI_List_1[613]  ;
	//  MesDataExd.MesData.AX_ProtectRelay_FeederMVCB[1].Mes20kVMidiSepamDefaultCablesOvercharge	:=	DI_List_1[641]  ;
	//  MesDataExd.MesData.AX_ProtectRelay_FeederMVCB[1].Mes20kVMidiHVCellDefaultFrom225kV			:=	DI_List_1[647]  ;
	MesDataExd.MesData.ProtectRelay_FeederMVCB[1].MesDataExd.MesData.MesTripped								:=	DI_List_1[738]  ;
	                                                                                	
	MesDataExd.MesData.ProtectRelay_FeederMVCB[2].MesDataExd.MesData.MesAlarmImax							:=	 DI_List_1[761] ;
	MesDataExd.MesData.ProtectRelay_FeederMVCB[2].MesAlarm_MaxP									:=   DI_List_1[763] ;
	MesDataExd.MesData.ProtectRelay_FeederMVCB[2].MesAlarm_Ground									:=   DI_List_1[765] ;  
	//  MesDataExd.MesData.AX_ProtectRelay_FeederMVCB[2].Mes20kVMidiSepamDefaultCablesOvercharge	:=   DI_List_1[793] ;
	//  MesDataExd.MesData.AX_ProtectRelay_FeederMVCB[2].Mes20kVMidiHVCellDefaultFrom225kV			:=   DI_List_1[799] ;
	MesDataExd.MesData.ProtectRelay_FeederMVCB[2].MesDataExd.MesData.MesTripped								:=   DI_List_1[890] ;
	
	MesDataExd.MesData.TapChanger.MesAlarm  := DI_List_1[1065] ;
	
	MesDataExd.MesData.MesAuxHTSect225kV							:=	DI_List_1[1217]	 ;
	MesDataExd.MesData.MesAuxHtSmaltHTBOpen						:=	DI_List_1[1219]	 ;
	MesDataExd.MesData.MesAuxHtFusionFuseMeasures225kV			:=	DI_List_1[1225]	 ;
	MesDataExd.MesData.MesAuxHtFusionFuseProtect225kV				:=	DI_List_1[1226]	 ;
	MesDataExd.MesData.MesAuxHtFusionFuseCountRte225kV			:=	DI_List_1[1227]	 ;
	MesDataExd.MesData.MesAuxHtShortCircuitCurrentProtectCcp2		:=	DI_List_1[1228]	 ;
	MesDataExd.MesData.MesAuxHtDisjCount20kVOpen					:=	DI_List_1[1230]	 ;
	MesDataExd.MesData.MesAuxHtDisjRefVoltage20kVOpen				:=	DI_List_1[1231]	 ;
	MesDataExd.MesData.MesAuxHtShortCircuitCurrentProtectCcp3		:=	DI_List_1[1232]	 ;
	MesDataExd.MesData.MesAuxBtTriggerGeneralDisj					:=	DI_List_1[1372]	 ;
	MesDataExd.MesData.MesAuxBt400VManqueAC						:=	DI_List_1[1373]	 ;
	MesDataExd.MesData.MesAuxBt400VDecltAntenneScada				:=	DI_List_1[1374]  ;
	MesDataExd.MesData.MesAuxBt400VDecltAntennePrio				:=	DI_List_1[1375]	 ;
	MesDataExd.MesData.MesAuxBt400VPermutAutoStopMode				:=	DI_List_1[1377]	 ;
	MesDataExd.MesData.MesAuxBt400VPermutAutoNormalMode			:=	DI_List_1[1378]	 ;
	MesDataExd.MesData.MesAuxBt400VPermutAutoSecoursMode			:=	DI_List_1[1379]	 ;
	MesDataExd.MesData.MesAuxBt400VPermutModeAuto					:=	DI_List_1[1380]	 ;
	MesDataExd.MesData.MesAuxBt400VVoltageLossNormalAlim			:=	DI_List_1[1381]	 ;
	MesDataExd.MesData.MesAuxBt400VVoltageLossSecoursAlim			:=	DI_List_1[1382]	 ;
	MesDataExd.MesData.MesAuxBt400VDefaultPermut					:=	DI_List_1[1383]	 ;
	
	
	
	MesDataExd.MesData.UPS_CE.MesAlarm_Batt 						:=	DI_List_1[1384]	 ;
	MesDataExd.MesData.UPS_CE.MesDataExd.MesData.MesAlarmState 				:=	DI_List_1[1385]	 ;
	MesDataExd.MesData.UPS_CE.MesAlarm_IsolBatt					:=	DI_List_1[1386]	 ;
	MesDataExd.MesData.UPS_CE.MesOpened_CBRectifier				:=	DI_List_1[1387]	 ;
	MesDataExd.MesData.UPS_CE.MesOpened_CBBatt					:=	DI_List_1[1388]	 ;
	MesDataExd.MesData.UPS_CE.MesOpened_CBAntenna					:=	DI_List_1[1389]	 ;
	MesDataExd.MesData.UPS_TCM.MesAlarm_Batt						:=	DI_List_1[1390]	 ;
	MesDataExd.MesData.UPS_TCM.MesDataExd.MesData.MesAlarmState				:=	DI_List_1[1391]	 ;
	MesDataExd.MesData.UPS_TCM.MesOpened_CBRectifier				:=	DI_List_1[1392]	 ;
	MesDataExd.MesData.UPS_TCM.MesOpened_CBBatt	   				:=	DI_List_1[1393]	 ;
	MesDataExd.MesData.UPS_TCM.MesOpened_CBAntenna				:=	DI_List_1[1394]	 ;
	 
	MesDataExd.MesData.MesAuxBtDefaultInverter					:=	DI_List_1[1395]	 ;
	MesDataExd.MesData.MesAuxBtSyntDefaultDistrib48VccJdb			:=	DI_List_1[1397]	 ;
	MesDataExd.MesData.MesAuxBtSyntOpenDistrib48VccJdb			:=	DI_List_1[1398]	 ;
	MesDataExd.MesData.MesAuxBtSyntDefaultDistrib48VccLocker		:=	DI_List_1[1403]	 ;
	MesDataExd.MesData.MesAuxBtSyntOpenDistrib48VccLocker			:=	DI_List_1[1404]	 ;
	 
	MesDataExd.MesData.Transfo_Aux.MesDataExd.MesData.MesAlarmTemp			:=	DI_List_1[1522]	 ;
	MesDataExd.MesData.Transfo_Aux.MesDataExd.MesData.MesAlarmGas			:=	DI_List_1[1523]	 ;
	MesDataExd.MesData.Transfo_Aux.MesDataExd.MesData.MesAlarmOilLevel		:=	DI_List_1[1524]	 ;
	 
	MesDataExd.MesData.MesAuxTransfoMeltingFusesContact			:=	DI_List_1[1525]	 ;                             
	MesDataExd.MesData.MesAuxTransfoSwitchGear	            	:=	DI_List_1[1526]  ;
	
	MesDataExd.MesData.DS.MesAlarmState          	  	:=	DI_List_1[1673] ;
	MesDataExd.MesData.FSS.MesAlarmFire				:=	DI_List_1[1674]	;
	MesDataExd.MesData.MesLocalRemoteOperation  	:=	DI_List_1[1682]	;
	MesDataExd.MesData.ES.MesAlarmState         		:=	DI_List_1[1683]	;
	 
	
						
	 /  MesDataExd.MesData.ProtectRelay_MainHVCB.MesDataExd.MesData.MesWatchdog 	  := DI_List_2[1]	; 
	MesDataExd.MesData.ProtectRelay_MainHVCB.MesDataExd.MesData.MesAlarmTCS    := DI_List_2[12]	;
	
	MesDataExd.MesData.ProtectRelay_Transfo225kV.MesDataExd.MesData.MesAlarmTCS 	 := DI_List_2[39] ;
	 // Mes225kVTransfoDefaultInternDisjCde := DI_List_2[46] ;
	
	MesDataExd.MesData.ProtectRelay_MainMVCB.MesDataExd.MesData.MesWatchdog 	 :=   DI_List_2[97]	; 
	MesDataExd.MesData.ProtectRelay_MainMVCB.MesDataExd.MesData.MesAlarmTCS   := 	DI_List_2[108]	;
	
	MesDataExd.MesData.ProtectRelay_FeederMVCB[1].MesDataExd.MesData.MesWatchdog   :=   DI_List_2[129] ;
	MesDataExd.MesData.ProtectRelay_FeederMVCB[1].MesDataExd.MesData.MesAlarmTCS   := 	 DI_List_2[140] ;
	
	MesDataExd.MesData.ProtectRelay_FeederMVCB[2].MesDataExd.MesData.MesWatchdog	  :=   DI_List_2[161]  ; 
	MesDataExd.MesData.ProtectRelay_FeederMVCB[2].MesDataExd.MesData.MesAlarmTCS   := 	 DI_List_2[172]  ;
	
	MesDataExd.MesData.TapChanger.MesAlarm_Discordance				  :=  DI_List_2[225]	;
	MesDataExd.MesData.TapChanger.MesAlarm_NoOutletDetected			  :=  DI_List_2[226]	;          
	MesDataExd.MesData.TapChanger.MesModeAuto							  :=  DI_List_2[227]	;
	MesDataExd.MesData.TapChanger.MesModeManual						  :=  DI_List_2[228]	;
	MesDataExd.MesData.TapChanger.MesState_ManoeuverAuthorized 		  :=  DI_List_2[230]	;
	
	MesDataExd.MesData.ProtectRelay_MainHVCB.OUT_CmdOpen  			  :=  DI_List_2[990] ;
	MesDataExd.MesData.ProtectRelay_MainHVCB.OUT_CmdClose     		  :=  DI_List_2[991] ;
	
	//  MesDataExd.MesData.Mes225kVTransfoDeclenchOpen	 := DI_List_2[1019] ;
	//  MesDataExd.MesData.Mes225kVTransfoEnclenchClose    := DI_List_2[1020] ;
	
	MesDataExd.MesData.ProtectRelay_MainMVCB.OUT_CmdOpen 	 :=  DI_List_2[1077] ;
	MesDataExd.MesData.ProtectRelay_MainMVCB.OUT_CmdClose  :=  DI_List_2[1078] ;
	
	MesDataExd.MesData.ProtectRelay_FeederMVCB[1].OUT_CmdOpen 	:=	DI_List_2[1106]  ; // MIDI 
	MesDataExd.MesData.ProtectRelay_FeederMVCB[1].OUT_CmdClose :=  DI_List_2[1107]  ;
	
	MesDataExd.MesData.ProtectRelay_FeederMVCB[2].OUT_CmdOpen   :=  DI_List_2[1135]	;	// PLAT 
	MesDataExd.MesData.ProtectRelay_FeederMVCB[2].OUT_CmdClose  :=  DI_List_2[1136]  ;
	
	MesDataExd.MesData.TapChanger.OUT_CmdRampUp	:=  DI_List_2[1193] ;
	MesDataExd.MesData.TapChanger.OUT_CmdRampDown :=	DI_List_2[1194] ;           
	MesDataExd.MesData.TapChanger.MesModeManual	:=  DI_List_2[1195]	;
	MesDataExd.MesData.TapChanger.MesModeAuto    :=  DI_List_2[1196] ;
	
	MesDataExd.MesData.MesAuxHtOpenSectLine225kV		  :=  DI_List_1[1242]  	;
	MesDataExd.MesData.MesAuxHtCloseSectLine225kV		  :=  DI_List_1[1243] 	;
	MesDataExd.MesData.MesAuxHtOpenSectMalt			  :=  DI_List_1[1244]   ;  
	MesDataExd.MesData.MesAuxHtCloseSectMalt			  :=  DI_List_1[1245]   ; 	
	MesDataExd.MesData.MesAuxHtTeleCondamnSl225kV		  :=  DI_List_1[1246] 	;
	MesDataExd.MesData.MesAuxHtDeTeleCondamnSl225kV	  :=  DI_List_1[1247]   ;                          
	MesDataExd.MesData.MesAuxHtTelecommandeRelestActif  :=  DI_List_1[1248]   ;
	MesDataExd.MesData.MesAuxHtTelecommandeRelestPassif :=  DI_List_1[1249]   ;
	
	//  MesDataExd.MesData.Filling Analogic Data			           
					                                
	MW(WORD_STRONG :=  AI_List_1[1  ],	WORD_WEAK := AI_List_1[1  ], SIZE := 1, FIX := 0, SIGNED := 0, VAR_OUT	:= MesDataExd.MesData.ProtectRelay_MainHVCB.MesDataExd.MesData.MesI1);
	MW(WORD_STRONG :=  AI_List_1[2  ],	WORD_WEAK := AI_List_1[2  ], SIZE := 1, FIX := 0, SIGNED := 0, VAR_OUT	:= MesDataExd.MesData.ProtectRelay_MainHVCB.MesDataExd.MesData.MesI2);
	MW(WORD_STRONG :=  AI_List_1[3  ],	WORD_WEAK := AI_List_1[3  ], SIZE := 1, FIX := 0, SIGNED := 0, VAR_OUT	:= MesDataExd.MesData.ProtectRelay_MainHVCB.MesDataExd.MesData.MesI3);
	MW(WORD_STRONG :=  AI_List_1[12 ],	WORD_WEAK := AI_List_1[12 ], SIZE := 1, FIX := 3, SIGNED := 0, VAR_OUT	:= MesDataExd.MesData.ProtectRelay_MainHVCB.MesDataExd.MesData.MesU12);
	MW(WORD_STRONG :=  AI_List_1[13 ],	WORD_WEAK := AI_List_1[13 ], SIZE := 1, FIX := 3, SIGNED := 0, VAR_OUT	:= MesDataExd.MesData.ProtectRelay_MainHVCB.MesDataExd.MesData.MesU23);
	MW(WORD_STRONG :=  AI_List_1[14 ],	WORD_WEAK := AI_List_1[14 ], SIZE := 1, FIX := 3, SIGNED := 0, VAR_OUT	:= MesDataExd.MesData.ProtectRelay_MainHVCB.MesDataExd.MesData.MesU31);
	MW(WORD_STRONG :=  AI_List_1[18 ],	WORD_WEAK := AI_List_1[18 ], SIZE := 1, FIX := 0, SIGNED := 0, VAR_OUT	:= MesDataExd.MesData.ProtectRelay_MainHVCB.MesU0);
	MW(WORD_STRONG :=  AI_List_1[21 ],	WORD_WEAK := AI_List_1[21 ], SIZE := 1, FIX := 0, SIGNED := 0, VAR_OUT	:= MesDataExd.MesData.ProtectRelay_MainHVCB.MesDataExd.MesData.MesFreq);
	MW(WORD_STRONG :=  AI_List_1[22 ],	WORD_WEAK := AI_List_1[22 ], SIZE := 1, FIX := 0, SIGNED := 0, VAR_OUT	:= MesDataExd.MesData.ProtectRelay_MainHVCB.MesP);
	MW(WORD_STRONG :=  AI_List_1[23 ],	WORD_WEAK := AI_List_1[23 ], SIZE := 1, FIX := 0, SIGNED := 0, VAR_OUT	:= MesDataExd.MesData.ProtectRelay_MainHVCB.MesQ);
	MW(WORD_STRONG :=  AI_List_1[27 ],	WORD_WEAK := AI_List_1[27 ], SIZE := 1, FIX := 0, SIGNED := 0, VAR_OUT	:= MesDataExd.MesData.ProtectRelay_MainHVCB.MesCosPhi);
	                               
	MW(WORD_STRONG :=  AI_List_1[33 ],	WORD_WEAK := AI_List_1[33 ], SIZE := 1, FIX := 0, SIGNED := 0, VAR_OUT	:= MesDataExd.MesData.ProtectRelay_Transfo225kV.MesDataExd.MesData.MesI1);
	MW(WORD_STRONG :=  AI_List_1[34 ],	WORD_WEAK := AI_List_1[34 ], SIZE := 1, FIX := 0, SIGNED := 0, VAR_OUT	:= MesDataExd.MesData.ProtectRelay_Transfo225kV.MesDataExd.MesData.MesI2);
	MW(WORD_STRONG :=  AI_List_1[35 ],	WORD_WEAK := AI_List_1[35 ], SIZE := 1, FIX := 0, SIGNED := 0, VAR_OUT	:= MesDataExd.MesData.ProtectRelay_Transfo225kV.MesDataExd.MesData.MesI3);
	MW(WORD_STRONG :=  AI_List_1[44 ],	WORD_WEAK := AI_List_1[44 ], SIZE := 1, FIX := 3, SIGNED := 0, VAR_OUT	:= MesDataExd.MesData.ProtectRelay_Transfo225kV.MesDataExd.MesData.MesU12);
	MW(WORD_STRONG :=  AI_List_1[45 ],	WORD_WEAK := AI_List_1[45 ], SIZE := 1, FIX := 3, SIGNED := 0, VAR_OUT	:= MesDataExd.MesData.ProtectRelay_Transfo225kV.MesDataExd.MesData.MesU23);
	MW(WORD_STRONG :=  AI_List_1[46 ],	WORD_WEAK := AI_List_1[46 ], SIZE := 1, FIX := 3, SIGNED := 0, VAR_OUT	:= MesDataExd.MesData.ProtectRelay_Transfo225kV.MesDataExd.MesData.MesU31);
	MW(WORD_STRONG :=  AI_List_1[54 ],	WORD_WEAK := AI_List_1[54 ], SIZE := 1, FIX := 0, SIGNED := 0, VAR_OUT	:= MesDataExd.MesData.ProtectRelay_Transfo225kV.MesP);
	MW(WORD_STRONG :=  AI_List_1[55 ],	WORD_WEAK := AI_List_1[55 ], SIZE := 1, FIX := 0, SIGNED := 0, VAR_OUT	:= MesDataExd.MesData.ProtectRelay_Transfo225kV.MesQ);
	
	MW(WORD_STRONG :=  AI_List_1[65 ],	WORD_WEAK := AI_List_1[65 ], SIZE := 1, FIX := 0, SIGNED := 0, VAR_OUT	:= MesDataExd.MesData.Mes20kVCourNeutCuveI1);
	MW(WORD_STRONG :=  AI_List_1[69 ],	WORD_WEAK := AI_List_1[69 ], SIZE := 1, FIX := 0, SIGNED := 0, VAR_OUT	:= MesDataExd.MesData.Mes20kVCourNeutCuveResidualI);
	MW(WORD_STRONG :=  AI_List_1[92 ],	WORD_WEAK := AI_List_1[92 ], SIZE := 1, FIX := 0, SIGNED := 0, VAR_OUT	:= MesDataExd.MesData.Mes20kVCourNeutCuveDecltI1);
	MW(WORD_STRONG :=  AI_List_1[95 ],	WORD_WEAK := AI_List_1[95 ], SIZE := 1, FIX := 0, SIGNED := 0, VAR_OUT	:= MesDataExd.MesData.Mes20kVCourNeutCuveDecltI2);
	
	MW(WORD_STRONG :=  AI_List_1[97  ],	WORD_WEAK := AI_List_1[97  ], SIZE := 1, FIX := 0, SIGNED := 0, VAR_OUT	:= MesDataExd.MesData.ProtectRelay_MainMVCB.MesDataExd.MesData.MesI1);
	MW(WORD_STRONG :=  AI_List_1[98  ],	WORD_WEAK := AI_List_1[98  ], SIZE := 1, FIX := 0, SIGNED := 0, VAR_OUT	:= MesDataExd.MesData.ProtectRelay_MainMVCB.MesDataExd.MesData.MesI2);
	MW(WORD_STRONG :=  AI_List_1[99  ],	WORD_WEAK := AI_List_1[99  ], SIZE := 1, FIX := 0, SIGNED := 0, VAR_OUT	:= MesDataExd.MesData.ProtectRelay_MainMVCB.MesDataExd.MesData.MesI3);
	MW(WORD_STRONG :=  AI_List_1[108 ],	WORD_WEAK := AI_List_1[108 ], SIZE := 1, FIX := 3, SIGNED := 0, VAR_OUT	:= MesDataExd.MesData.ProtectRelay_MainMVCB.MesDataExd.MesData.MesU12);
	MW(WORD_STRONG :=  AI_List_1[109 ],	WORD_WEAK := AI_List_1[109 ], SIZE := 1, FIX := 3, SIGNED := 0, VAR_OUT	:= MesDataExd.MesData.ProtectRelay_MainMVCB.MesDataExd.MesData.MesU23);
	MW(WORD_STRONG :=  AI_List_1[110 ],	WORD_WEAK := AI_List_1[110 ], SIZE := 1, FIX := 3, SIGNED := 0, VAR_OUT	:= MesDataExd.MesData.ProtectRelay_MainMVCB.MesDataExd.MesData.MesU31);
	MW(WORD_STRONG :=  AI_List_1[114 ],	WORD_WEAK := AI_List_1[114 ], SIZE := 1, FIX := 0, SIGNED := 0, VAR_OUT	:= MesDataExd.MesData.ProtectRelay_MainMVCB.MesU0);
	MW(WORD_STRONG :=  AI_List_1[117 ],	WORD_WEAK := AI_List_1[117 ], SIZE := 1, FIX := 0, SIGNED := 0, VAR_OUT	:= MesDataExd.MesData.ProtectRelay_MainMVCB.MesDataExd.MesData.MesFreq);
	MW(WORD_STRONG :=  AI_List_1[119 ],	WORD_WEAK := AI_List_1[119 ], SIZE := 1, FIX := 0, SIGNED := 0, VAR_OUT	:= MesDataExd.MesData.ProtectRelay_MainMVCB.MesP);
	MW(WORD_STRONG :=  AI_List_1[120 ],	WORD_WEAK := AI_List_1[120 ], SIZE := 1, FIX := 0, SIGNED := 0, VAR_OUT	:= MesDataExd.MesData.ProtectRelay_MainMVCB.MesQ);
	MW(WORD_STRONG :=  AI_List_1[123 ],	WORD_WEAK := AI_List_1[123 ], SIZE := 1, FIX := 0, SIGNED := 0, VAR_OUT	:= MesDataExd.MesData.ProtectRelay_MainMVCB.MesCosPhi);
	
	MW(WORD_STRONG :=  AI_List_2[1 	 ], WORD_WEAK := AI_List_2[1 ], SIZE := 1, FIX := 0, SIGNED := 0, VAR_OUT	:= MesDataExd.MesData.ProtectRelay_FeederMVCB[1].MesDataExd.MesData.MesI1);
	MW(WORD_STRONG :=  AI_List_2[2   ], WORD_WEAK := AI_List_2[2 ], SIZE := 1, FIX := 0, SIGNED := 0, VAR_OUT	:= MesDataExd.MesData.ProtectRelay_FeederMVCB[1].MesDataExd.MesData.MesI2);
	MW(WORD_STRONG :=  AI_List_2[3   ], WORD_WEAK := AI_List_2[3 ], SIZE := 1, FIX := 0, SIGNED := 0, VAR_OUT	:= MesDataExd.MesData.ProtectRelay_FeederMVCB[1].MesDataExd.MesData.MesI3);
	MW(WORD_STRONG :=  AI_List_2[22  ], WORD_WEAK := AI_List_2[22 ], SIZE := 1, FIX := 0, SIGNED := 0, VAR_OUT	:= MesDataExd.MesData.ProtectRelay_FeederMVCB[1].MesP);
	MW(WORD_STRONG :=  AI_List_2[23  ], WORD_WEAK := AI_List_2[23 ], SIZE := 1, FIX := 0, SIGNED := 0, VAR_OUT	:= MesDataExd.MesData.ProtectRelay_FeederMVCB[1].MesQ);
	                                                        
	MW(WORD_STRONG :=  AI_List_2[33 ], WORD_WEAK := AI_List_2[33 ], SIZE := 1, FIX := 0, SIGNED := 0, VAR_OUT	:= MesDataExd.MesData.ProtectRelay_FeederMVCB[2].MesDataExd.MesData.MesI1);
	MW(WORD_STRONG :=  AI_List_2[34 ], WORD_WEAK := AI_List_2[34 ], SIZE := 1, FIX := 0, SIGNED := 0, VAR_OUT	:= MesDataExd.MesData.ProtectRelay_FeederMVCB[2].MesDataExd.MesData.MesI2);
	MW(WORD_STRONG :=  AI_List_2[35 ], WORD_WEAK := AI_List_2[35 ], SIZE := 1, FIX := 0, SIGNED := 0, VAR_OUT	:= MesDataExd.MesData.ProtectRelay_FeederMVCB[2].MesDataExd.MesData.MesI3);
	MW(WORD_STRONG :=  AI_List_2[54 ], WORD_WEAK := AI_List_2[54 ], SIZE := 1, FIX := 0, SIGNED := 0, VAR_OUT	:= MesDataExd.MesData.ProtectRelay_FeederMVCB[2].MesP);         
	MW(WORD_STRONG :=  AI_List_2[55 ], WORD_WEAK := AI_List_2[55 ], SIZE := 1, FIX := 0, SIGNED := 0, VAR_OUT	:= MesDataExd.MesData.ProtectRelay_FeederMVCB[2].MesQ);         

END_IF
//MW(WORD_STRONG :=  AI_List_2[97 ], WORD_WEAK := AI_List_2[97 ], SIZE := 1, FIX := 0, SIGNED := 0, VAR_OUT	:= MesDataExd.MesData.Mes20kVPlatSepamQ);	






(*			
//  MesDataExd.MesData.Filling Digital Data				

MesData.Mes225kVCombiDefaultPhase1			:= DI_List_1[1]   ;
MesData.Mes225kVCombiDefaultPhase2		    := DI_List_1[2]   ;
MesData.Mes225kVCombiDefaultPhase3			:= DI_List_1[3]   ;
MesData.Mes225kVCombiDefaultPhaseRpt		:= DI_List_1[33]  ;
MesData.Mes225kVCombiDefaultGround			:= DI_List_1[35]  ;
MesData.Mes225kVCombiDefaultGroundRpt		:= DI_List_1[36]  ;
MesData.Mes225kVCombiDefaultMaxUInverse		:= DI_List_1[37]  ;
MesData.Mes225kVCombiDefaultMaxP			:= DI_List_1[38]  ;
MesData.Mes225kVCombiDefaultCircuitbreaker	:= DI_List_1[39]  ;	
MesData.Mes225kVCombiDefaultWatchdog		:= DI_List_1[148] ;
			
MesDataExd.MesData.Mes225kVTransfoDiscordSectLigneHTB		   := DI_List_1[164]    ;
MesDataExd.MesData.Mes225kVTransfoDiscordSectMaltHTB         := DI_List_1[165]    ;
MesDataExd.MesData.Mes225kVTransfoDiscordSectDisjHTB         := DI_List_1[166]    ;
MesDataExd.MesData.Mes225kVTransfoTeleCondamne               := DI_List_1[167]    ;
MesDataExd.MesData.Mes225kVTransfoDeTeleCondamne             := DI_List_1[168]    ;
MesDataExd.MesData.Mes225kVTransfoDiscordTeleCondamne	       := DI_List_1[169]    ;
MesDataExd.MesData.Mes225kVTransfoMaxI	                   := DI_List_1[170]    ;
MesDataExd.MesData.Mes225kVTransfoMaxICoteProd               := DI_List_1[171]    ;
MesDataExd.MesData.Mes225kVTransfoMaxIoCoteProd              := DI_List_1[172]    ;
MesDataExd.MesData.Mes225kVTransfoMinU                       := DI_List_1[173]    ;
MesDataExd.MesData.Mes225kVTransfoMinULong                   := DI_List_1[174]    ;
MesDataExd.MesData.Mes225kVTransfoMaxU                       := DI_List_1[175]    ;
MesDataExd.MesData.Mes225kVTransfoMaxULong                   := DI_List_1[176]    ;
MesDataExd.MesData.Mes225kVTransfoDefaultPhaseRpt            := DI_List_1[177]    ;
MesDataExd.MesData.Mes225kVTransfoAlarmImgTherm              := DI_List_1[178]    ;
MesDataExd.MesData.Mes225kVTransfoDefaultImgTherm            := DI_List_1[179]    ;
MesDataExd.MesData.Mes225kVTransfoDifferTransfo              := DI_List_1[180]    ;
MesDataExd.MesData.Mes225kVTransfoMaxFreq                    := DI_List_1[181]    ;
MesDataExd.MesData.Mes225kVTransfoMinFreq                    := DI_List_1[183]    ;
MesDataExd.MesData.Mes225kVTransfoCircuitBreaker             := DI_List_1[193]    ;
MesDataExd.MesData.Mes225kVTransfoDisjManqueSf6              := DI_List_1[197]    ;
MesDataExd.MesData.Mes225kVTransfoCmdDisjDesarm              := DI_List_1[198]    ;
MesDataExd.MesData.Mes225kVTransfoCmdDisjDistVerr            := DI_List_1[199]    ;
MesDataExd.MesData.Mes225kVTransfoDefaultMoteurArm           := DI_List_1[200]    ;
MesDataExd.MesData.Mes225kVTransfoDefaultAux230Vac           := DI_List_1[201]    ;
MesDataExd.MesData.Mes225kVTransfoDefaultAlimBobine          := DI_List_1[202]    ;
MesDataExd.MesData.Mes225kVTransfoAlarmBuchholz              := DI_List_1[220]    ;
MesDataExd.MesData.Mes225kVTransfoTriggerBuchHolz            := DI_List_1[221]    ;
MesDataExd.MesData.Mes225kVTransfoAlarmTempOil               := DI_List_1[222]    ;
MesDataExd.MesData.Mes225kVTransfoTriggerTempOil             := DI_List_1[223]    ;
MesDataExd.MesData.Mes225kVTransfoImgTherm1erStade           := DI_List_1[224]    ;
MesDataExd.MesData.Mes225kVTransfoImgTherm2emeStade          := DI_List_1[225]    ;
MesDataExd.MesData.Mes225kVTransfoDcltSurpression            := DI_List_1[228]    ;
MesDataExd.MesData.Mes225kVTransfoNiveauMiniOil              := DI_List_1[229]    ;
MesDataExd.MesData.Mes225kVTransfoRefrigLocal                := DI_List_1[230]    ;
MesDataExd.MesData.Mes225kVTransfoDcltClapetAntiRetour       := DI_List_1[231]    ;
MesDataExd.MesData.Mes225kVTransfoDcltRelaisProtectRegl      := DI_List_1[232]    ;
MesDataExd.MesData.Mes225kVTransfoDefaillanceRegl            := DI_List_1[233]    ;

MesDataExd.MesData.Mes20kVCourNeutCuveDefaultMasseCuve1		:= DI_List_1[305]	;
MesDataExd.MesData.Mes20kVCourNeutCuveMaxIexp2				:= DI_List_1[306]   ;
MesDataExd.MesData.Mes20kVCourNeutCuveDefaultMasseCuve2  		:= DI_List_1[307]   ;
MesDataExd.MesData.Mes20kVCourNeutCuveMaxIexp4				:= DI_List_1[308]   ;
MesDataExd.MesData.Mes20kVCourNeutCuveDefaultGround	    	:= DI_List_1[309]   ;
MesDataExd.MesData.Mes20kVCourNeutCuveMaxI0exp4		    	:= DI_List_1[310]   ;
MesDataExd.MesData.Mes20kVCourNeutCuveTempAlarm		    	:= DI_List_1[439]   ;
MesDataExd.MesData.Mes20kVCourNeutCuveTempTrigger				:= DI_List_1[440]   ;
MesDataExd.MesData.Mes20kVCourNeutCuveGazDischarge			:= DI_List_1[441]   ;
MesDataExd.MesData.Mes20kVCourNeutCuvePressure           		:= DI_List_1[442]   ;

MesDataExd.MesData.Mes20kVGeneralSepamDefaultPhase1			:= DI_List_1[457]	;
MesDataExd.MesData.Mes20kVGeneralSepamDefaultPhase2			:= DI_List_1[459]   ;
MesDataExd.MesData.Mes20kVGeneralHVCellDefaultCircuitBreaker	:= DI_List_1[495]   ;
MesDataExd.MesData.Mes20kVGeneralHVCellProtectCircuitBreaker	:= DI_List_1[586]   ;
MesDataExd.MesData.Mes20kVGeneralHVCellDefaultFrom225kV		:= DI_List_1[592]   ;

MesDataExd.MesData.Mes20kVMidiSepamDefaultShortCircuit		:=	DI_List_1[609]	;
MesDataExd.MesData.Mes20kVMidiSepamDefaultOvercharge			:=	DI_List_1[611]  ;
MesDataExd.MesData.Mes20kVMidiSepamDefaultGround				:=	DI_List_1[613]  ;
MesDataExd.MesData.Mes20kVMidiSepamDefaultCablesOvercharge	:=	DI_List_1[641]  ;
MesDataExd.MesData.Mes20kVMidiHVCellDefaultFrom225kV			:=	DI_List_1[647]  ;
MesDataExd.MesData.Mes20kVMidiHVCellProtectCircuitBreaker		:=	DI_List_1[738]  ;

MesDataExd.MesData.Mes20kVPlatSepamDefaultShortCircuit		:=	 DI_List_1[761] ;
MesDataExd.MesData.Mes20kVPlatSepamDefaultOvercharge		 	:=   DI_List_1[763] ;
MesDataExd.MesData.Mes20kVPlatSepamDefaultGround			 	:=   DI_List_1[765] ;  
MesDataExd.MesData.Mes20kVPlatSepamDefaultCablesOvercharge	:=   DI_List_1[793] ;
MesDataExd.MesData.Mes20kVPlatHVCellDefaultFrom225kV		 	:=   DI_List_1[799] ;
MesDataExd.MesData.Mes20kVPlatHVCellProtectCircuitBreaker     :=   DI_List_1[890] ;

MesDataExd.MesData.Mes225kVRegleurDefault := DI_List_1[1065] ;

MesDataExd.MesData.MesAuxHTSect225kV							:=	DI_List_1[1217]	 ;
MesDataExd.MesData.MesAuxHtSmaltHTBOpen						:=	DI_List_1[1219]	 ;
MesDataExd.MesData.MesAuxHtFusionFuseMeasures225kV			:=	DI_List_1[1225]	 ;
MesDataExd.MesData.MesAuxHtFusionFuseProtect225kV				:=	DI_List_1[1226]	 ;
MesDataExd.MesData.MesAuxHtFusionFuseCountRte225kV			:=	DI_List_1[1227]	 ;
MesDataExd.MesData.MesAuxHtShortCircuitCurrentProtectCcp2		:=	DI_List_1[1228]	 ;
MesDataExd.MesData.MesAuxHtDisjCount20kVOpen					:=	DI_List_1[1230]	 ;
MesDataExd.MesData.MesAuxHtDisjRefVoltage20kVOpen				:=	DI_List_1[1231]	 ;
MesDataExd.MesData.MesAuxHtShortCircuitCurrentProtectCcp3		:=	DI_List_1[1232]	 ;
MesDataExd.MesData.MesAuxBtTriggerGeneralDisj					:=	DI_List_1[1372]	 ;
MesDataExd.MesData.MesAuxBt400VManqueAC						:=	DI_List_1[1373]	 ;
MesDataExd.MesData.MesAuxBt400VDecltAntenneScada				:=	DI_List_1[1374]  ;
MesDataExd.MesData.MesAuxBt400VDecltAntennePrio				:=	DI_List_1[1375]	 ;
MesDataExd.MesData.MesAuxBt400VPermutAutoStopMode				:=	DI_List_1[1377]	 ;
MesDataExd.MesData.MesAuxBt400VPermutAutoNormalMode			:=	DI_List_1[1378]	 ;
MesDataExd.MesData.MesAuxBt400VPermutAutoSecoursMode			:=	DI_List_1[1379]	 ;
MesDataExd.MesData.MesAuxBt400VPermutModeAuto					:=	DI_List_1[1380]	 ;
MesDataExd.MesData.MesAuxBt400VVoltageLossNormalAlim			:=	DI_List_1[1381]	 ;
MesDataExd.MesData.MesAuxBt400VVoltageLossSecoursAlim			:=	DI_List_1[1382]	 ;
MesDataExd.MesData.MesAuxBt400VDefaultPermut					:=	DI_List_1[1383]	 ;
MesDataExd.MesData.MesAuxBt48VCeDefaultBatt					:=	DI_List_1[1384]	 ;
MesDataExd.MesData.MesAuxBt48VCeDefaultRedress				:=	DI_List_1[1385]	 ;
MesDataExd.MesData.MesAuxBt48VCeDefaultIsolBatt				:=	DI_List_1[1386]	 ;
MesDataExd.MesData.MesAuxBt48VCeDecltDisjRedress				:=	DI_List_1[1387]	 ;
MesDataExd.MesData.MesAuxBt48VCeDecltDisjBatt					:=	DI_List_1[1388]	 ;
MesDataExd.MesData.MesAuxBt48VCeDecltAntenne					:=	DI_List_1[1389]	 ;
MesDataExd.MesData.MesAuxBt48VTcmDefaultBatt					:=	DI_List_1[1390]	 ;
MesDataExd.MesData.MesAuxBt48VTcmDefaultRedress				:=	DI_List_1[1391]	 ;
MesDataExd.MesData.MesAuxBt48VTcmDecltDisjRedress				:=	DI_List_1[1392]	 ;
MesDataExd.MesData.MesAuxBt48VTcmDecltDisjBatt				:=	DI_List_1[1393]	 ;
MesDataExd.MesData.MesAuxBt48VTcmDecltAntenne					:=	DI_List_1[1394]	 ;
MesDataExd.MesData.MesAuxBtDefaultInverter					:=	DI_List_1[1395]	 ;
MesDataExd.MesData.MesAuxBtSyntDefaultDistrib48VccJdb			:=	DI_List_1[1397]	 ;
MesDataExd.MesData.MesAuxBtSyntOpenDistrib48VccJdb			:=	DI_List_1[1398]	 ;
MesDataExd.MesData.MesAuxBtSyntDefaultDistrib48VccLocker		:=	DI_List_1[1403]	 ;
MesDataExd.MesData.MesAuxBtSyntOpenDistrib48VccLocker			:=	DI_List_1[1404]	 ;
MesDataExd.MesData.MesAuxTransfoTempTrigger					:=	DI_List_1[1522]	 ;
MesDataExd.MesData.MesAuxTransfoGazDischarge					:=	DI_List_1[1523]	 ;
MesDataExd.MesData.MesAuxTransfoPressure						:=	DI_List_1[1524]	 ;
MesDataExd.MesData.MesAuxTransfoMeltingFusesContact			:=	DI_List_1[1525]	 ;                             
MesDataExd.MesData.MesAuxTransfoSwitchGear	            	:=	DI_List_1[1526]  ;

MesDataExd.MesData.MesPDLDoorsOpen         	  	:=	DI_List_1[1673]	;
MesDataExd.MesData.MesPDLFireDetectorSystem    	:=	DI_List_1[1674]	;
MesDataExd.MesData.MesPDLLocalRemoteOperation  	:=	DI_List_1[1682]	;
MesDataExd.MesData.MesPDLEmergencyStop         	:=	DI_List_1[1683]	;
					
MesDataExd.MesData.Mes225kVCombiWatchdog		 := DI_List_2[1]	; 
MesDataExd.MesData.Mes225kVCombiDefaultMajor   := DI_List_2[12]	;

MesDataExd.MesData.Mes225kVTransfoSepamMajorDefault	 := DI_List_2[39] ;
MesDataExd.MesData.Mes225kVTransfoDefaultInternDisjCde := DI_List_2[46] ;

MesDataExd.MesData.Mes20kVGeneralSepamWatchdog	   :=   DI_List_2[97]	; 
MesDataExd.MesData.Mes20kVGeneralSepamDefaultMajor   := 	DI_List_2[108]	;

MesDataExd.MesData.Mes20kVMidiSepamWatchdog		:=   DI_List_2[129] ;
MesDataExd.MesData.Mes20kVMidiSepamDefaultMajor   := 	 DI_List_2[140] ;

MesDataExd.MesData.Mes20kVPlatSepamWatchdog		:=   DI_List_2[161]  ; 
MesDataExd.MesData.Mes20kVPlatSepamDefaultMajor   := 	 DI_List_2[172]  ;

MesDataExd.MesData.Mes225kVRegleurDefaultDiscordance	:=  DI_List_2[225]	;
MesDataExd.MesData.Mes225kVRegleurNoOutletDetected	:=	DI_List_2[226]	;          
MesDataExd.MesData.Mes225kVRegleurRegleurModeAuto		:=	DI_List_2[227]	;
MesDataExd.MesData.Mes225kVRegleurRegleurModeManuel	:=  DI_List_2[228]	;
MesDataExd.MesData.Mes225kVRegleurManoeuverAuthorized :=  DI_List_2[230]	;

MesDataExd.MesData.Mes225kVCombiOrderOpenCircuitBreaker 	:=  DI_List_2[990] ;
MesDataExd.MesData.Mes225kVCombiOrderCloseCircuitBreaker  :=  DI_List_2[991] ;

MesDataExd.MesData.Mes225kVTransfoDeclenchOpen	 := DI_List_2[1019] ;
MesDataExd.MesData.Mes225kVTransfoEnclenchClose    := DI_List_2[1020] ;

MesDataExd.MesData.Mes20kVGeneralHVCellProtectOrderOpenCircuitBreaker	 :=  DI_List_2[1077] ;
MesDataExd.MesData.Mes20kVGeneralHVCellProtectOrderCloseCircuitBreaker :=  DI_List_2[1078] ;

MesDataExd.MesData.Mes20kVMidiHVCellProtectOrderOpenCircuitBreaker	:=	DI_List_2[1106]  ;
MesDataExd.MesData.Mes20kVMidiHVCellProtectOrderCloseCircuitBreaker   :=  DI_List_2[1107]  ;

MesDataExd.MesData.Mes20kVPlatHVCellProtectOrderOpenCircuitBreaker   :=  DI_List_2[1135]	;
MesDataExd.MesData.Mes20kVPlatHVCellProtectOrderCloseCircuitBreaker  :=  DI_List_2[1136]  ;

MesDataExd.MesData.Mes225kVRegleurCdeMontee	:=  DI_List_2[1193] ;
MesDataExd.MesData.Mes225kVRegleurCdeDescente :=	DI_List_2[1194] ;           
MesDataExd.MesData.Mes225kVRegleurModeManuel	:=  DI_List_2[1195]	;
MesDataExd.MesData.Mes225kVRegleurModeAuto    :=  DI_List_2[1196] ;

MesDataExd.MesData.MesAuxHtOpenSectLine225kV		  :=  DI_List_1[1242]  	;
MesDataExd.MesData.MesAuxHtCloseSectLine225kV		  :=  DI_List_1[1243] 	;
MesDataExd.MesData.MesAuxHtOpenSectMalt			  :=  DI_List_1[1244]   ;  
MesDataExd.MesData.MesAuxHtCloseSectMalt			  :=  DI_List_1[1245]   ; 	
MesDataExd.MesData.MesAuxHtTeleCondamnSl225kV		  :=  DI_List_1[1246] 	;
MesDataExd.MesData.MesAuxHtDeTeleCondamnSl225kV	  :=  DI_List_1[1247]   ;                          
MesDataExd.MesData.MesAuxHtTelecommandeRelestActif  :=  DI_List_1[1248]   ;
MesDataExd.MesData.MesAuxHtTelecommandeRelestPassif :=  DI_List_1[1249]   ;

//  MesDataExd.MesData.Filling Analogic Data			           
				                                
MW(WORD_STRONG :=  AI_List_1[1  ],	WORD_WEAK := AI_List_1[1  ], SIZE := 1, FIX := 0, SIGNED := 0, VAR_OUT	:= MesDataExd.MesData.Mes225kVCombiI1);
MW(WORD_STRONG :=  AI_List_1[2  ],	WORD_WEAK := AI_List_1[2  ], SIZE := 1, FIX := 0, SIGNED := 0, VAR_OUT	:= MesDataExd.MesData.Mes225kVCombiI2);
MW(WORD_STRONG :=  AI_List_1[3  ],	WORD_WEAK := AI_List_1[3  ], SIZE := 1, FIX := 0, SIGNED := 0, VAR_OUT	:= MesDataExd.MesData.Mes225kVCombiI3);
MW(WORD_STRONG :=  AI_List_1[12 ],	WORD_WEAK := AI_List_1[12 ], SIZE := 1, FIX := 3, SIGNED := 0, VAR_OUT	:= MesDataExd.MesData.Mes225kVCombiU21);
MW(WORD_STRONG :=  AI_List_1[13 ],	WORD_WEAK := AI_List_1[13 ], SIZE := 1, FIX := 3, SIGNED := 0, VAR_OUT	:= MesDataExd.MesData.Mes225kVCombiU32);
MW(WORD_STRONG :=  AI_List_1[14 ],	WORD_WEAK := AI_List_1[14 ], SIZE := 1, FIX := 3, SIGNED := 0, VAR_OUT	:= MesDataExd.MesData.Mes225kVCombiU13);
MW(WORD_STRONG :=  AI_List_1[18 ],	WORD_WEAK := AI_List_1[18 ], SIZE := 1, FIX := 0, SIGNED := 0, VAR_OUT	:= MesDataExd.MesData.Mes225kVCombiResidualU);
MW(WORD_STRONG :=  AI_List_1[21 ],	WORD_WEAK := AI_List_1[21 ], SIZE := 1, FIX := 0, SIGNED := 0, VAR_OUT	:= MesDataExd.MesData.Mes225kVCombiFrequency);
MW(WORD_STRONG :=  AI_List_1[22 ],	WORD_WEAK := AI_List_1[22 ], SIZE := 1, FIX := 0, SIGNED := 0, VAR_OUT	:= MesDataExd.MesData.Mes225kVCombiP);
MW(WORD_STRONG :=  AI_List_1[23 ],	WORD_WEAK := AI_List_1[23 ], SIZE := 1, FIX := 0, SIGNED := 0, VAR_OUT	:= MesDataExd.MesData.Mes225kVCombiQ);
MW(WORD_STRONG :=  AI_List_1[27 ],	WORD_WEAK := AI_List_1[27 ], SIZE := 1, FIX := 0, SIGNED := 0, VAR_OUT	:= MesDataExd.MesData.Mes225kVCombiCosPhi);
                               
MW(WORD_STRONG :=  AI_List_1[33 ],	WORD_WEAK := AI_List_1[33 ], SIZE := 1, FIX := 0, SIGNED := 0, VAR_OUT	:= MesDataExd.MesData.Mes225kVTransfoI1);
MW(WORD_STRONG :=  AI_List_1[34 ],	WORD_WEAK := AI_List_1[34 ], SIZE := 1, FIX := 0, SIGNED := 0, VAR_OUT	:= MesDataExd.MesData.Mes225kVTransfoI2);
MW(WORD_STRONG :=  AI_List_1[35 ],	WORD_WEAK := AI_List_1[35 ], SIZE := 1, FIX := 0, SIGNED := 0, VAR_OUT	:= MesDataExd.MesData.Mes225kVTransfoI3);
MW(WORD_STRONG :=  AI_List_1[44 ],	WORD_WEAK := AI_List_1[44 ], SIZE := 1, FIX := 3, SIGNED := 0, VAR_OUT	:= MesDataExd.MesData.Mes225kVTransfoU21);
MW(WORD_STRONG :=  AI_List_1[45 ],	WORD_WEAK := AI_List_1[45 ], SIZE := 1, FIX := 3, SIGNED := 0, VAR_OUT	:= MesDataExd.MesData.Mes225kVTransfoU32);
MW(WORD_STRONG :=  AI_List_1[46 ],	WORD_WEAK := AI_List_1[46 ], SIZE := 1, FIX := 3, SIGNED := 0, VAR_OUT	:= MesDataExd.MesData.Mes225kVTransfoU13);
MW(WORD_STRONG :=  AI_List_1[54 ],	WORD_WEAK := AI_List_1[54 ], SIZE := 1, FIX := 0, SIGNED := 0, VAR_OUT	:= MesDataExd.MesData.Mes225kVTransfoP);
MW(WORD_STRONG :=  AI_List_1[55 ],	WORD_WEAK := AI_List_1[55 ], SIZE := 1, FIX := 0, SIGNED := 0, VAR_OUT	:= MesDataExd.MesData.Mes225kVTransfoQ);

MW(WORD_STRONG :=  AI_List_1[65 ],	WORD_WEAK := AI_List_1[65 ], SIZE := 1, FIX := 0, SIGNED := 0, VAR_OUT	:= MesDataExd.MesData.Mes20kVCourNeutCuveI1);
MW(WORD_STRONG :=  AI_List_1[69 ],	WORD_WEAK := AI_List_1[69 ], SIZE := 1, FIX := 0, SIGNED := 0, VAR_OUT	:= MesDataExd.MesData.Mes20kVCourNeutCuveResidualI);
MW(WORD_STRONG :=  AI_List_1[92 ],	WORD_WEAK := AI_List_1[92 ], SIZE := 1, FIX := 0, SIGNED := 0, VAR_OUT	:= MesDataExd.MesData.Mes20kVCourNeutCuveDecltI1);
MW(WORD_STRONG :=  AI_List_1[95 ],	WORD_WEAK := AI_List_1[95 ], SIZE := 1, FIX := 0, SIGNED := 0, VAR_OUT	:= MesDataExd.MesData.Mes20kVCourNeutCuveDecltI2);

MW(WORD_STRONG :=  AI_List_1[97  ],	WORD_WEAK := AI_List_1[97  ], SIZE := 1, FIX := 0, SIGNED := 0, VAR_OUT	:= MesDataExd.MesData.Mes20kVGeneralSepamI1);
MW(WORD_STRONG :=  AI_List_1[98  ],	WORD_WEAK := AI_List_1[98  ], SIZE := 1, FIX := 0, SIGNED := 0, VAR_OUT	:= MesDataExd.MesData.Mes20kVGeneralSepamI2);
MW(WORD_STRONG :=  AI_List_1[99  ],	WORD_WEAK := AI_List_1[99  ], SIZE := 1, FIX := 0, SIGNED := 0, VAR_OUT	:= MesDataExd.MesData.Mes20kVGeneralSepamI3);
MW(WORD_STRONG :=  AI_List_1[108 ],	WORD_WEAK := AI_List_1[108 ], SIZE := 1, FIX := 3, SIGNED := 0, VAR_OUT	:= MesDataExd.MesData.Mes20kVGeneralSepamU21);
MW(WORD_STRONG :=  AI_List_1[109 ],	WORD_WEAK := AI_List_1[109 ], SIZE := 1, FIX := 3, SIGNED := 0, VAR_OUT	:= MesDataExd.MesData.Mes20kVGeneralSepamU32);
MW(WORD_STRONG :=  AI_List_1[110 ],	WORD_WEAK := AI_List_1[110 ], SIZE := 1, FIX := 3, SIGNED := 0, VAR_OUT	:= MesDataExd.MesData.Mes20kVGeneralSepamU13);
MW(WORD_STRONG :=  AI_List_1[114 ],	WORD_WEAK := AI_List_1[114 ], SIZE := 1, FIX := 0, SIGNED := 0, VAR_OUT	:= MesDataExd.MesData.Mes20kVGeneralSepamResidualU);
MW(WORD_STRONG :=  AI_List_1[117 ],	WORD_WEAK := AI_List_1[117 ], SIZE := 1, FIX := 0, SIGNED := 0, VAR_OUT	:= MesDataExd.MesData.Mes20kVGeneralSepamFrequency);
MW(WORD_STRONG :=  AI_List_1[119 ],	WORD_WEAK := AI_List_1[119 ], SIZE := 1, FIX := 0, SIGNED := 0, VAR_OUT	:= MesDataExd.MesData.Mes20kVGeneralSepamP);
MW(WORD_STRONG :=  AI_List_1[120 ],	WORD_WEAK := AI_List_1[120 ], SIZE := 1, FIX := 0, SIGNED := 0, VAR_OUT	:= MesDataExd.MesData.Mes20kVGeneralSepamQ);
MW(WORD_STRONG :=  AI_List_1[123 ],	WORD_WEAK := AI_List_1[123 ], SIZE := 1, FIX := 0, SIGNED := 0, VAR_OUT	:= MesDataExd.MesData.Mes20kVGeneralSepamCosPhi);

MW(WORD_STRONG :=  AI_List_2[1 	 ], WORD_WEAK := AI_List_2[1 ], SIZE := 1, FIX := 0, SIGNED := 0, VAR_OUT	:= MesDataExd.MesData.Mes20kVMidiSepamI1);
MW(WORD_STRONG :=  AI_List_2[2   ], WORD_WEAK := AI_List_2[2 ], SIZE := 1, FIX := 0, SIGNED := 0, VAR_OUT	:= MesDataExd.MesData.Mes20kVMidiSepamI2);
MW(WORD_STRONG :=  AI_List_2[3   ], WORD_WEAK := AI_List_2[3 ], SIZE := 1, FIX := 0, SIGNED := 0, VAR_OUT	:= MesDataExd.MesData.Mes20kVMidiSepamI3);
MW(WORD_STRONG :=  AI_List_2[22  ], WORD_WEAK := AI_List_2[22 ], SIZE := 1, FIX := 0, SIGNED := 0, VAR_OUT	:= MesDataExd.MesData.Mes20kVMidiSepamP);
MW(WORD_STRONG :=  AI_List_2[23  ], WORD_WEAK := AI_List_2[23 ], SIZE := 1, FIX := 0, SIGNED := 0, VAR_OUT	:= MesDataExd.MesData.Mes20kVMidiSepamQ);
                                                        
MW(WORD_STRONG :=  AI_List_2[33 ], WORD_WEAK := AI_List_2[33 ], SIZE := 1, FIX := 0, SIGNED := 0, VAR_OUT	:= MesDataExd.MesData.Mes20kVPlatSepamI1);
MW(WORD_STRONG :=  AI_List_2[34 ], WORD_WEAK := AI_List_2[34 ], SIZE := 1, FIX := 0, SIGNED := 0, VAR_OUT	:= MesDataExd.MesData.Mes20kVPlatSepamI2);
MW(WORD_STRONG :=  AI_List_2[35 ], WORD_WEAK := AI_List_2[35 ], SIZE := 1, FIX := 0, SIGNED := 0, VAR_OUT	:= MesDataExd.MesData.Mes20kVPlatSepamI3);
MW(WORD_STRONG :=  AI_List_2[54 ], WORD_WEAK := AI_List_2[54 ], SIZE := 1, FIX := 0, SIGNED := 0, VAR_OUT	:= MesDataExd.MesData.Mes20kVPlatSepamP);
MW(WORD_STRONG :=  AI_List_2[55 ], WORD_WEAK := AI_List_2[55 ], SIZE := 1, FIX := 0, SIGNED := 0, VAR_OUT	:= MesDataExd.MesData.Mes20kVPlatSepamQ);

MW(WORD_STRONG :=  AI_List_2[97 ], WORD_WEAK := AI_List_2[97 ], SIZE := 1, FIX := 0, SIGNED := 0, VAR_OUT	:= MesDataExd.MesData.Mes20kVPlatSepamQ);


*)
END_METHOD

END_FUNCTION_BLOCK

// ---- 01_Equipement_Library/PCS/FB_PCS_Base.TcPOU
FUNCTION_BLOCK FB_PCS_Base
//////////////////
// PCS controller . Base FB
//////////////////

VAR_INPUT PERSISTENT
	// Parameters of the Object (instance specific) 
	ParamUnitID 					: BYTE  	:= 1; 			  		(* (NA)   CTRLPcs Modbus Unit ID.*)
	ParamIPAddress			   		: STRING ; 		(* (NA) Config IP Adress of CTRLPCs*)
	ParamIPAddress_DSP				: ARRAY[1..3] OF  STRING ; 			(* (NA) DSP IP Address*)
	ParamTcpPort					: UINT		:= 502;					(* (NA) Modbus TCP Port*)
	ParamNbPowerCol					: BYTE	 	:= 4 ; 					(* (NA) Config : Number of Pcs/Module controlled . *)
                                                                
	ParamTempoComAlarm				: TIME 		:= T#5S ; 				(* (s) Config : Tempo to detect LOC Alarm*)
	ParamTempoComWarning			: TIME 		:= T#5S ; 				(* (s) Config : Tempo to detect LOC Alarm*)
	ParamTimeOutBlckStrt			: TIME 		:= T#3M ;				(* (s) Config : Tempo to start before Timeout warning*)

	ParamClockReadTime 				: TIME 		:= TIME#200MS;	  		(* (Time) Read Modbus Frequency .   *)
	ParamClockWriteTime 			: TIME 		:= TIME#200MS;   		(* (Time) Write Modbus Frequency .         *)
	ParamTimeout					: TIME  	:= T#1S ;		  		(* (Time) Timeout for modbus reading*)
	                                                                	
	ParamTimePulseTrig				: TIME 		:= T#10S;            	(* (Time)Pulse duration for commands *)		
	                                                                	
	ParamEssNum						: UINT 		:= 1;					(* (NA) ID number of the Pcs' father PCS*)
	ParamPcsNum						: UINT 		:= 1;					(* (NA) ID number of the PCS *)
END_VAR

VAR_OUTPUT
	//Child objects
	
END_VAR

VAR_INPUT
	// I/O Inputs 
		// ALARM MANAGEMENT //
		IN_SetptP					: REAL ;						// (kW)   [P,H] Dynamic aCtive Power  setpoint 
		IN_SetptQ					: REAL ;						// (kVAr) [P,H] Dynamic reactive Power setpoint 
		testP : REAL;
		testQ : REAL;
		IN_SetptU					: REAL ;						// (kW)   [P,H] Dynamic active Power  setpoint 
		IN_SetptF					: REAL ;						// (kW)   [P,H] Dynamic active Power  setpoint 
		IN_SetptCosPhi				: REAL;							// (NA)  [P,H] Dynamic CosPhi setpoint	
		
		{attribute 'OPC.UA.DA' := '1'} 
		IN_SetptP_Local						: REAL;				// Local Command
		{attribute 'OPC.UA.DA' := '1'} 
		IN_SetptQ_Local						: REAL;				// Local Command
		{attribute 'OPC.UA.DA' := '1'} 
		IN_CmdReset							: BOOL ;
		{attribute 'OPC.UA.DA' := '1'} 
		IN_CmdStandby						: BOOL;				// Cmd To send a soft Stop (No opening and closing of the AC/DC switch )
		{attribute 'OPC.UA.DA' := '1'} 
		IN_CmdStart							: BOOL;				// Cmd To send a start to the PCS (Does the full procedure, Soft + Close AC + Close DC)
		{attribute 'OPC.UA.DA' := '1'} 
		IN_CmdStop							: BOOL;				// Cmd To send a stop to the PCS (Soft Stop + Open DC + Open AC)
			                            
		
		IN_CmdToggleRead					: BOOL;
        IN_CmdToggleWrite					: BOOL;

		

		
		IN_CmdPcsInLocalMode		 		: BOOL ; 




END_VAR

VAR
	//M_ALARMMANAGEMENT VARIABLES//
		TON_ComAlarm				: TON ; 			// Tempo before deteting loss of communication. 
		TON_ComWarning				: TON ; 			// Tempo before deteting loss of communication. 
                                         

		MesComWarning				: BOOL ; 			// (NA) [P,H]   True if bad communication 
		MesComAlarm					: BOOL ; 			// (NA) True if complete loss of modbus communication 

	//M_CP VARIABLES//
		Trig_Cmd_Read				: R_TRIG;                                                                                        
		Trig_Cmd_Write				: R_TRIG;                                                                                        
        
	//M_READ VARIABLES//
	///MesDataExd	AT%Q*		: PCS ;											// (NA) [P,H,B] CTRLPcs  Data Structure
		
	//M_WRITECOMMAND VARIABLES//


	//M_STATEMANAGER VARIABLES//
		MesState					: BYTE ; 						// (NA) [P,H,B] Bit0: 1 = Not Available (AC or DC breaker open or AllAcContactorsOpened), Bit1: GridMode: 1=grid	
	
	//M_WRITESETPOINTS VARIABLES//
	
		FB_CheckSetpt1				: FB_CheckSetpt ; 				// (NA) Functionnal Block to check if active power Writing Successful
		FB_CheckSetpt2				: FB_CheckSetpt ; 				// (NA) Functionnal Block to check if reactive power Writing Successful

	//M_INIT VARIABLES //
		bInit						: BOOL 			:= TRUE ; 		// (NA) Initialize object parameters at first cycle 
		
	// M_EXECUTE VARIABLES //
		TP1							: TP ; 						// (NA) Tempo to define Modbus Reading Frequency 
		TP2 						: TP ; 						// (NA) Tempo to define Modbus Writing Frequency
                                    
		ClockRead		AT%Q*		: BOOL;							// (NA) Modbus reading Clock
		TrigRead 					: R_TRIG;							// (NA) Modbus writing Clock 	
		ClockWrite 		AT%Q*		: BOOL;							// (NA) Modbus writing Clock 	
		TrigWrite 					: R_TRIG;							// (NA) Modbus writing Clock 	
		CalCP_Start                 : BOOL ; 						// (NA) Permanent conditions to activate method
		CalCP_Stop                  : BOOL ;                       	// (NA) Permanent conditions to activate method   	
	    CalCP_Reset                 : BOOL ; 						// (NA) Permanent conditions to activate method  

		CalCP_Standby 				: BOOL ; 						// (NA) Permanent conditions to activate method  


		MesCP_Read					: BOOL := TRUE;	(* Read function enable *)
		MesCP_Write					: BOOL := FALSE;	(* Write function enable *)	
		
		
END_VAR

METHOD M_AlarmManagement
//////////////////
//  PCS Alarm Management 
/////////////////

VAR 
	// Method local variables (reinitialized at each cycle) 

	
END_VAR
END_METHOD

METHOD M_CP
//////////////////
//  Permanent Condition 
/////////////////

VAR 
	// Method local variables (reinitialized at each cycle) 
	
END_VAR
END_METHOD

METHOD M_Evaluate : BOOL
VAR_INPUT
END_VAR
END_METHOD

METHOD M_Execute
//////////////////
//  Method Calls 
/////////////////

VAR 
	// Method local variables (reinitialized at each cycle) 
	KK			: BYTE;			// For Loop 
	
END_VAR
// READING AND WRITING CLOCK //
	TP1(IN:=NOT TP1.Q , PT:= ParamClockReadTime);
	TrigRead(CLK :=	TP1.Q );
	ClockRead 		:=TrigRead.Q ;
	
	TP2(IN:=NOT TP2.Q , PT:= ParamClockWriteTime);
	TrigWrite(CLK :=	TP2.Q );
	ClockWrite 		:= TrigWrite.Q;
	
// PERMANENT CONDITIONS //
	M_CP() ; 

// METHODS CALLS //
	IF bInit THEN
		M_Init() ; 
		bInit					:= FALSE ; 
	ELSIF CmdInit_G THEN 
		bInit:= TRUE ;
		
	END_IF

	M_Read() ; 
	M_Evaluate();                                                               
	M_StateManager() ;
	M_WriteSetPoints() ; 
	M_WriteCommand() ; 
	
// COM MANAGER //


	M_AlarmManagement();
END_METHOD

METHOD M_Init

VAR 

END_VAR
END_METHOD

METHOD M_Read
//////////////////
//  Read Modbus Variable for PCS . 
/////////////////

VAR 
	// Method local variables (reinitialized at each cycle) 


END_VAR
END_METHOD

METHOD M_StateManager
//////////////////
// Detect which is the state of the PCS system . 
/////////////////

VAR 
	// Method local variables (reinitialized at each cycle) 

	
END_VAR
	
// OPERATIONNAL INDEX //
END_METHOD

METHOD M_WriteCommand
//////////////////
//  Modbus Write of the command for the PCS. 
/////////////////

VAR 
	// Method local variables (reinitialized at each cycle) 
		
END_VAR
END_METHOD

METHOD M_WriteSetPoints
//////////////////
//  Modbus Write of the active and reactive power setpoints of the PCS . 
/////////////////
VAR 
	// Method local variables (reinitialized at each cycle) 

END_VAR
END_METHOD

END_FUNCTION_BLOCK

// ---- 01_Equipement_Library/PCS/FB_PCS_Jema_IBX3.TcPOU
FUNCTION_BLOCK FB_PCS_Jema_IBX3 EXTENDS FB_PCS_Base
//////////////////
// PLC controller . Jema Object 
//////////////////

VAR_INPUT PERSISTENT
	// Parameters of the Object
		ParamPn							: REAL := 1500.0;		(* (kW) Nominal power*)
		ParamQn							: REAL := 1500.0;		(* (kW) Nominal power*)
		ParamSn								: REAL := 1500.0;	(* (kVA) Maximum apparent power of the PCS (lasts 30s)*)
		
		ParamTimeoutCmdQ					: TIME := T#15S; 	(* (s) Time to activate or deactivate Q regulation before an alarm is raised*)
		ParamTimeoutCmdCosPhi				: TIME := T#15S; 	(* (s) Time to activate or deactivate CosPhi regulation before an alarm is raised*)
		ParamTimeoutQvU						: TIME := T#15S;	(* (s) Time to activate or deactivate Q(U) regulation before an alarm is raised*)
		ParamTimeoutPvF						: TIME := T#15S;	(* (s) Time to activate or deactivate P(f) regulation before an alarm is raised*)
		ParamTimeOutBat						: TIME := T#1M;		(* (ms) Battery alarm time before a soft stop is sent to the equipment*)
		ParamTimeoutGridFormerTransition	: TIME := T#1M ;	(* (ms) Time elapsed after grid former cmd when an alarm is raised*)
		ParamTimeoutGridFeederTransition	: TIME := T#1M;		(* (ms) Time elapsed after grid feeder cmd when an alarm is raised*)
 		ParamTimeoutOffTransition			: TIME := T#1M;		// (ms) Time elapsed after CmdStop cmd when an alarm is raised
   	
    {attribute 'OPC.UA.DA' := '1'}                		
		ParamAllowRechargeLowSoc			: BOOL := TRUE;		(* (NA) if true, the PCS will charge when SoC between Soc_Min and Soc_Stop*)
    {attribute 'OPC.UA.DA' := '1'}                		
		ParamPrechargeLowSoc				: REAL := 30;		(* (kW) setpoint sent at low SoC*)
    {attribute 'OPC.UA.DA' := '1'}                		
		ParamTimeLowSocToRecharge			: TIME := T#5M;		(* (ms) Time elapsed in low soc area before a soft stop is sent again *)
		ParamPoverQ							: BOOL := TRUE;		// If P over Q is True, then Max setpoint for Q calculated from setpoint of P
    	          	
		ParamQfU_UDbHigh    				: REAL;				(* (V) JEMA U1 : AKUO U_UDbHigh*)
		ParamQfU_Umax		    			: REAL;				(* (V) JEMA U2 : AKUO U_Umax*)
		ParamQfU_UDbLow	    				: REAL;				(* (V) JEMA U3 : AKUO U_UDbLow*)
		ParamQfU_Umin		    			: REAL;				(* (V) JEMA U4 : AKUO U_Umin*)
		                            		
		ParamQfU_QDbHigh					: REAL;				(* (kVAr) JEMA Q1 : AKUO U_QDbHigh*)
		ParamQfU_Qmax						: REAL;				(* (kVAr) JEMA Q2 : AKUO U_Qmax*)
		ParamQfU_QDbLow						: REAL;				(* (kVAr) JEMA Q3 : AKUO U_QDbLow*)
		ParamQfU_Qmin						: REAL;				(* (kVAr) JEMA Q4 : AKUO U_Qmin*)
    	                            		
		ParamPfF_FDbHigh	    			: REAL;				(* (Hz) JEMA f1 : AKUO P_FDbHigh*)
		ParamPfF_Fmax		    			: REAL;				(* (Hz) JEMA f2 : AKUO P_Fmax*)
		ParamPfF_FDbLow	    				: REAL;				(* (Hz) JEMA f3 : AKUO P_FDbLow*)
		ParamPfF_Fmin		    			: REAL;				(* (Hz) JEMA f4 : AKUO P_Fmin*)
		                            		
		ParamPfF_PDbHigh					: REAL;				(* (kW) JEMA P1 : AKUO P_PDbHigh*)
		ParamPfF_Pmax						: REAL;				(* (kW) JEMA P2 : AKUO P_Pmax*)
		ParamPfF_PDbLow						: REAL;				(* (kW) JEMA P3 : AKUO P_PDbLow*)
		ParamPfF_Pmin						: REAL;				(* (kW) JEMA P4 : AKUO P_Pmin*)
    	
		ParamPfF_FhystLow					: REAL;				(* (Hz) JEMA fst1*)
		ParamPfF_FhystHigh					: REAL;				(* (Hz) JEMA fst2*)
		
		ParamFLow_droop						: REAL;				(* (Hz) flow frequency (droop curve)*)
		ParamFHigh_droop					: REAL;				(* (Hz) fhigh frequency (droop curve)*)
		ParamULow_droop						: REAL;				(* (V) Ulow voltage (droop curve)*)
		ParamUHigh_droop					: REAL;				(* (V) Ulow voltage (droop curve)*)
		
		ParamTimeSoCRangeReachedRmp			: TIME;				(* (ms) Time to ramp P back to the setpoint after the SoC reached its limits*)
		ParamTimeFreqRegStbDuration			: TIME;				(* (ms) Time to ramp P back to the setpoint after entering the stable *)
		ParamTimeEnterStblPriorRmp			: TIME; 			(* (ms) Time to wait after entering the stable before ramping the P back to the setpoint*)
    	                            	
		ParamFreqRegSoCmax 					: REAL;	 			(* (%) Jema Stops charging setpoint and overfreq regulation if BESS reaches this value*)
		ParamFreqRegSoCmin 					: REAL;				(* (%) Jema Stops discharging setpoint and underfreq regulation if BESS reaches this value*)

		ParamSetPtModbusMode				: BOOL := TRUE;		(* (NA) If True, then Setpoints come from Modbus*)    	
		ParamLVRT_Enabled					: BOOL; 			(* (NA) LVRT Enabled *)
		ParamAntiIslanding_Enabled			: BOOL;				(* (NA) Is Anti Islanding enabled*)
    {attribute 'OPC.UA.DA' := '1'}                		
		ParamDeactivateWatchdog				: BOOL := TRUE;				// Parameter to deactivate the watchdog

    {attribute 'OPC.UA.DA' := '1'}                		
		ParamSocLow							: REAL := 10;		(* (%) SoC from which we start limiting the maximal output Power*)
    {attribute 'OPC.UA.DA' := '1'}                		
		ParamSocHigh						: REAL := 85;		(* (%) SoC from which we start limiting the minimal output Power*)
    {attribute 'OPC.UA.DA' := '1'}                		
		ParamSocMin_G						: REAL := 5;		(* (%) Minimal SoC *)	
    {attribute 'OPC.UA.DA' := '1'}                		
		ParamSocMax_G						: REAL := 90;		(* (%) Maximal SoC *)	
    {attribute 'OPC.UA.DA' := '1'}                		
		ParamSocStop						: REAL := 3;		(* (%) SoC from which we stop the PCS*)
    {attribute 'OPC.UA.DA' := '1'}                		
		ParamSocRecharge					: REAL := 4;		(* (%) SoC from which we recharge the PCS*)	
    {attribute 'OPC.UA.DA' := '1'}                		
		ParamPCharge						: REAL := -10;		(* (kW) power at which we consider the PCS Recharges*)

    {attribute 'OPC.UA.DA' := '1'}                		
		ParamChargeEfficiency				: REAL := 97;		(* (%) percentage of efficiency of PCS during charge*)
    {attribute 'OPC.UA.DA' := '1'}                		
		ParamDischargeEfficiency			: REAL := 97;		(* (%) percentage of efficiency of PCS during discharge*)
		
END_VAR 
VAR_INPUT   	                   			
	MesDataExd								: PCS_Jema_IBX3 ;
	// Commands :
		IN_CmdPcsLocal						: BOOL;				// PCS is not included in available PCS' pool (excluded from HPP control). 
		IN_CmdStopOperation					: BOOL;				// BESS Specific command : Stop operation		
		IN_CmdPreventStart					: BOOL;				// BESS Specific command : Prevent start	
		IN_CmdOpenAC						: BOOL;				// Cmd To send an Open AC order
		IN_CmdOpenDC						: BOOL;				// Cmd To send an Open DC order	
 		IN_CmdP_On							: BOOL;				// Cmd start regulating on SetptP from outside of PCS : if you wan to know from what source, add a _IO2 value
		IN_CmdQ_On							: BOOL;				// Cmd start regulating on SetptQ from outside of PCS : if you wan to know from what source, add a _IO2 value
		IN_CmdCosPhi_On						: BOOL;				// Cmd start regulating on SetptCosPhi from outside of PCS : if you wan to know from what source, add a _IO2 value
		IN_CmdP_Off							: BOOL;				// Cmd start regulating on SetptP from outside of PCS : if you wan to know from what source, add a _IO2 value
		IN_CmdQ_Off							: BOOL;				// Cmd start regulating on SetptQ from outside of PCS : if you wan to know from what source, add a _IO2 value
		IN_CmdCosPhi_Off					: BOOL;				// Cmd start regulating on SetptCosPhi from outside of PCS : if you wan to know from what source, add a _IO2 value
		IN_CmdFreqregOn						: BOOL;				// Cmd 
		IN_CmdFreqregOff					: BOOL;				// 
		IN_CmdUregOn						: BOOL;				// 
		IN_CmdUregOff						: BOOL;				// 
	                      		
		IN_CmdBlackStart					: BOOL; 			// Cmd Black start from outside of PCS : if you wan to know from what source, add a _IO2 value
		IN_CmdGridFormer					: BOOL;				// 
		IN_CmdGridFeeder					: BOOL;				// 
	
		IN_SetptU_Local						: REAL := 500;	// Local Command
		IN_SetptF_Local						: REAL := 50;		// Local Command
		
		IN_CmdWatchdog						: BOOL ; 			// Activate or Deactivate the Watchdog function
	                
END_VAR
VAR_OUTPUT
	//Child objects
		OUT_SetptP_IO					: INT;			// (NA) Analogical value for the active power setpoint (based on ParamPnom)
		OUT_SetptQ_IO					: INT;			// (NA) Analogical value for the reactive power setpoint (based on ParamQnom)

END_VAR
VAR      
	MesPSetpt_Test : REAL;
	MesQSetpt_Test : REAL;    
                           	
	//M_ALARMMANAGEMENT VARIABLES//  
		AX_AlarmWords						: ARRAY[1..30] OF ST_ValuesAlarms;
		AX_AlarmWords_Null					: ARRAY[1..30] OF ST_ValuesAlarms;
		AX_AlarmWordsJema					: ARRAY[1..225] OF ST_ValuesAlarms;
		AX_AlarmWordsJema_Null				: ARRAY[1..225] OF ST_ValuesAlarms;
		NumAlarmsActive						: UINT;
		NumAlarmsActiveJema					: UINT;
		TON_BatComAlarm						: TON;
	//M_READ VARIABLES//            		
		TP_ReadCompleted					: TP;
		MesBlock1_Temp_Old					: ARRAY [1..4] OF ARRAY[1..120] OF WORD ; // (NA) Temporary Block Matrix for PCS modbus reading		

		ModbusRead            				: ARRAY [1..4] OF FB_ModbusRead ; 	// (NA) FB for Modbus Reading
		MesBlock1_Temp						: ARRAY [1..4] OF ARRAY[1..120] OF WORD ; // (NA) Temporary Block Matrix for PCS modbus reading		
		AX_PcsHeartbit						: ARRAY [1..4] OF BOOL;
		                                	
		MesModbusReadAlarm 		  			: ARRAY [1..4] OF BOOL ;				// (NA) Modbus Read Alarm for communication
		TON_PcsHeartBitAlarm				: ARRAY [1..4] OF TON ;	
		TON_AlarmPcs						: ARRAY [1..4] OF TON ; 			// DesInhibate undervoltage alarms on PCS few seconds after PCS connected .  
                                        	
		DFV									: ARRAY[1..3] OF FB_DetectFixedValue;	
		StaticValuesToCompareHeartbit		: ARRAY[1..3] OF REAL;
		                                	                                     
		CTU_PcsNb							: CTU ; 
	

	// M_EVALUATE VARIABLES//
		Time_Discharge_LowSoc				: TIME;
		Time_Start_Discharge_LowSoc			: TIME;
		MesStatusWatchdog					: BOOL;
		MesHeartbeat_Old					: WORD;
		Trig_Watchdog						: R_TRIG;
		DataSystemBMS						: BAT_SAMS;
		
	// Microcycling //
		MesMicroCyclingP					: REAL;				// (kW) Actual P for microcyling mode (if micro act = either ParamPmicro/-ParamPmicor, else 0)		
		MesMicroCyclingP_Old				: REAL;				// (kW) Active power the PCS will have during microcyling
	    MesMicroCyclingAllowed				: BOOL;				// (NA) If SoC is in range for microCycling                        		
		Trig_MicroCyclingNoLongerAllowed	: F_TRIG;			// Trig to detect falling edge of microcylingAllowed

	//M_WRITECOMMAND VARIABLES//    		
		ModbusWrite							: ARRAY [1..3] OF FB_ModbusWrite ;				// (NA) Functionnal Block for Writing Command Word through modbus
		Trig_Write							: ARRAY [1..3] OF R_TRIG;               		
		MesModbusWriteCmdAlarm				: ARRAY [1..3] OF BOOL ;						// (NA) Modbus Write Failed  (Command word) . 	
		MesModbusWriteCode          		: ARRAY [1..3] OF UDINT ; 						// (NA) Modbus Write Alarm Code 
		CmdWrite			AT%Q*			: ARRAY [1..3] OF BOOL;                     	
		AX_Cmd				AT%Q*			: ARRAY [1..3] OF ARRAY [1..120] OF WORD;   	
		AX_Cmd_Old							: ARRAY [1..3] OF ARRAY [1..120] OF WORD;   	
                                   		                                                	
		TRIG_CmdOpenAC						: R_TRIG;										// Trig to detect an order to change Mode
		TRIG_CmdOpenDC						: R_TRIG;										// Trig to detect an order to change Mode
		TRIG_CmdP_On						: R_TRIG;										// Trig to detect an order to change Mode
		TRIG_CmdQ_On			    		: R_TRIG;										// Trig to detect an order to change Mode
		TRIG_CmdCosPhi_On 					: R_TRIG;										// Trig to detect an order to change Mode
		TRIG_CmdP_Off						: R_TRIG;										// Trig to detect an order to change Mode
		TRIG_CmdQ_Off			    		: R_TRIG;										// Trig to detect an order to change Mode
		TRIG_CmdCosPhi_Off 					: R_TRIG;										// Trig to detect an order to change Mode
		TRIG_CmdBlackStart					: R_TRIG;										// Trig to detect an order to change Mode
		TRIG_CmdReset						: R_TRIG;		
		TRIG_FreqReg_On						: R_TRIG;
		TRIG_FreqReg_Off					: R_TRIG;
		TRIG_UReg_On						: R_TRIG;
		TRIG_UReg_Off						: R_TRIG;
		TRIG_CmdGridFormer					: R_TRIG;
		TRIG_CmdGridFeeder					: R_TRIG;
		TRIG_CmdMicroCyclingOn				: R_TRIG;
		TRIG_CmdMicroCyclingOff     		: R_TRIG;
		TRIG_CmdStop						: R_TRIG;
		TRIG_CmdStandby						: R_TRIG;
		TRIG_CmdStart						: R_TRIG;
		TRIG_CmdPcsLocal					: R_TRIG;
		
		TRIG_Recharge_LowSoc				: R_TRIG;
		TRIG_RechargeBackToNormalSoc		: R_TRIG;
		TRIG_SocStop						: R_TRIG;
		TON_SocStop							: TON;
		TRIG_SocStop_Again					: R_TRIG;
        TRIG_BackToNormalSoc				: R_TRIG;
                		
		TP_CmdBlackStart					: TP;				// TP To ensure R trig is detected
		TP_Reset							: TP ; 				// (NA) Maintain Reset command for a certain time 
		TP_CmdStandby						: TP;				// TP To maintain a soft stop order

		// Pour la commande start, j'envoie une consigne pour fermer les contacteurs DC des batteries
		TP_CmdOpenAC						: TP;				// TP To ensure R trig is detected
		TP_CmdOpenDC						: TP;				// TP To ensure R trig is detected

		TP_CmdStart							: TP;				// TP To ensure R trig is detected
		TP_CmdPreStart						: TP;				// TP To send a close dc breaker order before sending start order
		F_TrigPreStart						: F_TRIG;			// failing edge to detect end of TP;
		
		// Pour la commande stop, pour éviter qu'on ouvre tout d'un coup, je faire un pré stop pendant 1,5s où j'envoie un autre de standby
		TP_CmdStop							: TP;				// TP To ensure R trig is detected
		TP_CmdPreStop						: TP;				// TP to send a soft stop before sending a stop 
		F_TrigPreStop						: F_TRIG;			// failing edge to detect end of TP;
		                            		
		TON_CmdP_On							: TON;			// Trig to detect an order to change Mode
		TON_CmdQ_On			    			: TON;			// Trig to detect an order to change Mode
		TON_CmdCosPhi_On 					: TON;			// Trig to detect an order to change Mode
		TON_CmdP_Off						: TON;			// Trig to detect an order to change Mode
		TON_CmdQ_Off			    		: TON;			// Trig to detect an order to change Mode
		TON_CmdCosPhi_Off 					: TON;			// Trig to detect an order to change Mode
		TON_CmdBlackStart					: TON;			// Trig to detect an order to change Mode
		TON_FreqReg_On						: TON;
		TON_FreqReg_Off						: TON;
		TON_UReg_On							: TON;
		TON_UReg_Off						: TON;
		TON_CmdGridFormer					: TON;
		TON_CmdGridFeeder					: TON;
		TON_CmdMicroCyclingOn				: TON;
		TON_CmdMicroCyclingOff     			: TON;
		TON_CmdStart			    		: TON;
		TON_CmdStop	                		: TON;
		TON_CmdStandby		        		: TON;
		TON_TimeAllowedToRecharge			: TON;		// tempo pour s'assurer que si start dans le mode low SOC, on stop après 10min si pas de chargement
		

		RS_hystlimitmin						: RS;
		RS_hystlimitmax						: RS;
 		RS_hystlimitEnergyShifmin			: RS;
		RS_hystlimitEnergyShifmax			: RS;
		
		CalPmaxCorr_highSoC					: REAL;
		CalPminCorr_lowSoC					: REAL;
        	           	                            		
END_VAR

METHOD M_AlarmManagement
//////////////////
//  PCS Alarm Management 
/////////////////

VAR 
	// Method local variables (reinitialized at each cycle) 
	FB_AlarmCodeManager : FB_AlarmCodeManager ; 
	KK					: UINT;				// For Loop
	ComWarning			: BOOL;				// Aggregated Wcommunication warning
	ComAlarm			: BOOL;				// Aggregated communication Alarm
	
	CalAlarmPcsSynthesis: BOOL;
	LL					: UINT;
	ID_Journal			: UINT;
	WordTest			: WORD;
	MesNbMots			: UINT;
END_VAR
// COMMUNICATION //
	ComWarning 				:=  MesModbusReadAlarm[1] OR MesModbusReadAlarm[2] OR MesModbusReadAlarm[3] ;		
	ComAlarm				:=  MesModbusReadAlarm[1] AND MesModbusReadAlarm[2] AND MesModbusReadAlarm[3]  ;
		
	TON_ComAlarm(IN:= ComAlarm , PT:= ParamTempoComAlarm, Q=>MesComAlarm) ;	
	TON_ComWarning(IN := ComWarning, PT := ParamTempoComWarning, Q => MesComWarning);
	TON_BatComAlarm(IN := AX_ESS[ParamEssNum].AX_Bat[ParamPcsNum].MesDataExd.MesData.MesAlarmCom, PT := ParamTimeOutBat );	
	
	MesDataExd.MesData.MesAlarmCom		:= MesComAlarm ; 
	MesDataExd.MesData.MesWarningCom 	:= MesComWarning ; 
	

// PCS ALARM INHIBITION
FOR KK := 1 TO ParamNbPowerCol DO
	TON_AlarmPcs[KK](IN:=NOT MesDataExd.MesData.MesState.0, PT:= T#5S ) ;
	IF NOT TON_AlarmPcs[KK].Q THEN 
		MesDataExd.AX_PowerCol[KK].MesRegAlarm0.4 := FALSE ; 
		MesDataExd.AX_PowerCol[KK].MesRegAlarm0.7 := FALSE ; 
		MesDataExd.AX_PowerCol[KK].MesRegAlarm0.9 := FALSE ; 
		MesDataExd.AX_PowerCol[KK].MesRegAlarm0.11 := FALSE ; 
		MesDataExd.AX_PowerCol[KK].MesRegAlarm0.13 := FALSE ;			
	END_IF
	
	DFV[KK](IN_Addr := ADR(MesDataExd.AX_PowerCol[KK].MesHeartbit), IN_EmptyStruct := ADR(StaticValuesToCompareHeartbit[KK]) , IN_Size := SIZEOF(MesDataExd.AX_PowerCol[KK].MesHeartbit), IN_Duration := T#10S, OUT_bStatic => AX_PcsHeartbit[KK] ) ; 
	
END_FOR	


// SYNTHESES ALARMES //
CalAlarmPcsSynthesis := MesDataExd.AX_PowerCol[1].MesRegAlarm0 > 0
OR MesDataExd.AX_PowerCol[2].MesRegAlarm0 > 0
OR MesDataExd.AX_PowerCol[3].MesRegAlarm0 > 0
OR MesDataExd.AX_PowerCol[1].MesRegAlarm1 > 0
OR MesDataExd.AX_PowerCol[2].MesRegAlarm1 > 0
OR MesDataExd.AX_PowerCol[3].MesRegAlarm1 > 0
OR MesDataExd.AX_PowerCol[1].MesRegAlarm2 > 0
OR MesDataExd.AX_PowerCol[2].MesRegAlarm2 > 0
OR MesDataExd.AX_PowerCol[3].MesRegAlarm2 > 0
OR MesDataExd.AX_PowerCol[1].MesRegAlarm3 > 0
OR MesDataExd.AX_PowerCol[2].MesRegAlarm3 > 0
OR MesDataExd.AX_PowerCol[3].MesRegAlarm3 > 0
OR MesDataExd.AX_PowerCol[1].MesRegAlarm4 > 0
OR MesDataExd.AX_PowerCol[2].MesRegAlarm4 > 0
OR MesDataExd.AX_PowerCol[3].MesRegAlarm4 > 0 ;


// AlarmCode		
	FB_AlarmCodeManager(
		bAlarm1		:= CalAlarmPcsSynthesis		,								// Power columns Alarm Synthesis, at least one alarm active on power column
		bAlarm2		:= TON_CmdP_On.Q OR TON_CmdP_Off.Q,							// Timeout for CmdP order
		bAlarm3		:= TON_CmdQ_On.Q OR TON_CmdQ_Off.Q,							// Timeout for CmdQ order			
		bAlarm4		:= TON_BatComAlarm.Q,										// Communication alarm with Batteries : SoftStop order sent to PCS                           			    	
		bAlarm5		:= TON_CmdBlackStart.Q,                                     // Timeout for BlackStart order   			
		bAlarm6		:= TON_FreqReg_On.Q OR TON_FreqReg_Off.Q,                   // Timeout for Freq Regulation activation                            				
		bAlarm7		:= TON_UReg_On.Q OR TON_UReg_Off.Q,                         // Timeout for Voltage Regulation activation
		bAlarm8 	:= TON_CmdGridFormer.Q,                                     // Timeout for grid former activation
		bAlarm9		:= TON_CmdGridFeeder.Q,                                     // Timeout for grid feeder activation
		bAlarm10	:= TON_CmdMicroCyclingOn.Q OR TON_CmdMicroCyclingOff.Q,     // Timeout for MicroCycling
		bAlarm11	:= MesDataExd.MesData.MesAlarmCom,                          // Communication alarm : none of the Power Columns are responding 				
		bAlarm12	:= IN_CmdStart and IN_CmdPreventStart,                      // Start command received whilst forbidden to start			
		bAlarm13	:= FALSE,                                               	//			
		bAlarm14	:= FALSE,                                               	//		
		bAlarm15	:= FALSE,                                               	//		
		wAlarmCode	=>MesDataExd.MesData.MesAlarmCode);		                                		
		                                                                                 	
		
// WARNING CODE //
	FB_AlarmCodeManager(
		bAlarm1		:= MesComWarning, 									// Communication warning : At least one of the Power Columns are not responding 
		bAlarm2		:= MesDataExd.MesData.MesState.4,					// PCS switches off because of low SOC
		bAlarm3		:= MesDataExd.MesData.MesState.4 AND IN_CmdStart,	// Command start while low SOC state                                          
		bAlarm4		:= MesDataExd.MesData.MesState.3,					// PCS Tries recharging because of low SOC                                          
		bAlarm5		:= MesDataExd.AX_PowerCol[3].MesDeratingWord.0,  																								// Power Column 3 derating active due to temperature
		bAlarm6		:= MesDataExd.AX_PowerCol[1].MesDeratingWord.4 OR MesDataExd.AX_PowerCol[2].MesDeratingWord.4 OR MesDataExd.AX_PowerCol[3].MesDeratingWord.4,      	// At least one power column has a derating due to overvoltage
		bAlarm7		:= MesDataExd.AX_PowerCol[1].MesDeratingWord.5 OR MesDataExd.AX_PowerCol[2].MesDeratingWord.5 OR MesDataExd.AX_PowerCol[3].MesDeratingWord.5,      	// At least one power column has a derating due to undervoltage
		bAlarm8		:= MesDataExd.AX_PowerCol[1].MesDeratingWord.6 OR MesDataExd.AX_PowerCol[2].MesDeratingWord.6 OR MesDataExd.AX_PowerCol[3].MesDeratingWord.6,      	// At least one power column has a derating due to overfrequency
		bAlarm9		:= MesDataExd.AX_PowerCol[1].MesDeratingWord.7 OR MesDataExd.AX_PowerCol[2].MesDeratingWord.7 OR MesDataExd.AX_PowerCol[3].MesDeratingWord.7,      	// At least one power column has a derating due to underfrequency
		bAlarm10	:= MesDataExd.AX_PowerCol[1].MesDoorOpened,        	// Power column 1 cabinet door is opened
		bAlarm11	:= MesDataExd.AX_PowerCol[2].MesDoorOpened,        	// Power column 2 cabinet door is opened
		bAlarm12	:= MesDataExd.AX_PowerCol[3].MesDoorOpened,        	// Power column 3 cabinet door is opened
		bAlarm13	:= MesDataExd.AX_PowerCol[2].MesDeratingWord.0,  		           													//Power Column 2 derating active due to temperature
		bAlarm14	:= MesDataExd.AX_PowerCol[1].MesDeratingWord.0,  		           													//Power Column 1 derating active due to temperature
		bAlarm15	:=FALSE , // 
		wAlarmCode	=>MesDataExd.MesData.MesWarningCode);
		
